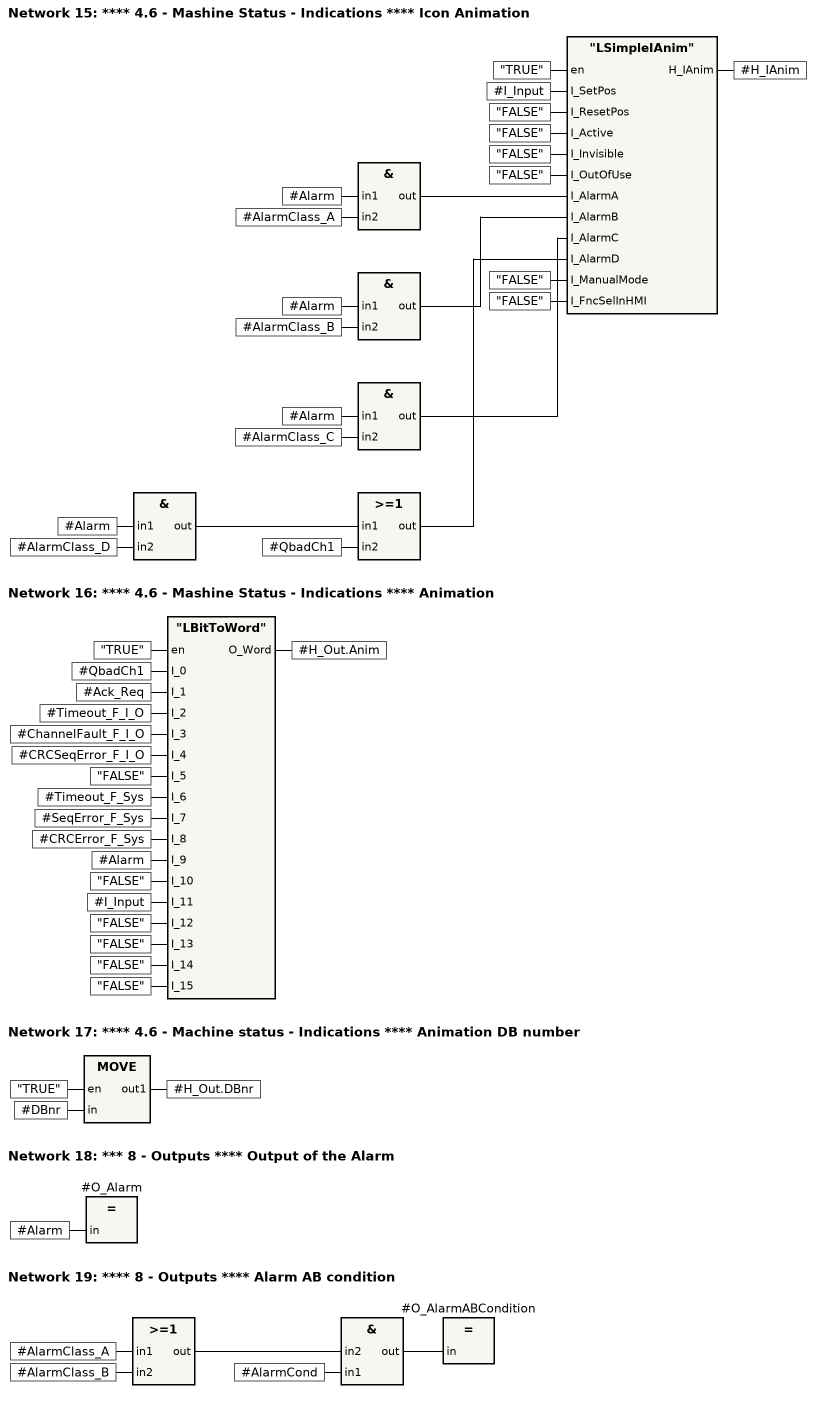
   IF "TRUE" THEN
       "LSimpleIAnim"(I_SetPos := #I_Input,
                      I_ResetPos := "FALSE",
                      I_Active := "FALSE",
                      I_Invisible := "FALSE",
                      I_OutOfUse := "FALSE",
                      I_AlarmA := #Alarm AND #AlarmClass_A,
                      I_AlarmB := #Alarm AND #AlarmClass_B,
                      I_AlarmC := #Alarm AND #AlarmClass_C,
                      I_AlarmD := (#Alarm AND #AlarmClass_D) OR #QbadCh1,
                      I_ManualMode := "FALSE",
                      I_FncSelInHMI := "FALSE",
                      H_IAnim => #H_IAnim);
   END_IF;
END_REGION

REGION Network 16: **** 4.6 - Mashine Status - Indications **** Animation
   // Animation
   IF "TRUE" THEN
       "LBitToWord"(I_0 := #QbadCh1,
                    I_1 := #Ack_Req,
                    I_2 := #Timeout_F_I_O,
                    I_3 := #ChannelFault_F_I_O,
                    I_4 := #CRCSeqError_F_I_O,
                    I_5 := "FALSE",
                    I_6 := #Timeout_F_Sys,
                    I_7 := #SeqError_F_Sys,
                    I_8 := #CRCError_F_Sys,
                    I_9 := #Alarm,
                    I_10 := "FALSE",
                    I_11 := #I_Input,
                    I_12 := "FALSE",
                    I_13 := "FALSE",
                    I_14 := "FALSE",
                    I_15 := "FALSE",
                    O_Word => #H_Out.Anim);
   END_IF;
END_REGION

REGION Network 17: **** 4.6 - Machine status - Indications **** Animation DB number
   // Animation DB number
   IF "TRUE" THEN #H_Out.DBnr := #DBnr; END_IF;
END_REGION

REGION Network 18: *** 8 - Outputs **** Output of the Alarm
   // Output of the Alarm
   #O_Alarm := #Alarm;
END_REGION

REGION Network 19: **** 8 - Outputs **** Alarm AB condition
   // Alarm AB condition
   #O_AlarmABCondition := (#AlarmClass_A OR #AlarmClass_B) AND #AlarmCond;
END_REGION
END_FUNCTION_BLOCK

FUNCTION_BLOCK "L1SafetyFbkAlarm"   // FB1422, FBD
TITLE = L1SafetyFbkAlarm
{ S7_Optimized_Access := 'FALSE' }
AUTHOR : VCC
FAMILY : AlarmHnd
NAME : 1SafeAlm
VERSION : 0.3
// ================================================================================
// TThis module evalute the diagnostic byte from the Siemens safety Functionblock 
// FB 216 "F_FDBACK" and generates a feedback alarm in the standard program.
// A boolean output is available to inform the upper level that the alarm can be 
// reset.
// This module generates also a word containing all necessary information for HMI 
// Icon animation, and a word with all information for HMI safety module 
// diagnostic screen. 
// ================================================================================
// stored: AutoNumber false, IsIECCheckEnabled false, SetENOAutomatically False, UDAEnableTagReadback false
   VAR_INPUT
      I_Feedback { ExternalAccessible := 'False'; ExternalVisible := 'False'; ExternalWritable := 'False'} : Bool;   // Input feedback
      I_AlarmClass { ExternalAccessible := 'False'; ExternalVisible := 'False'; ExternalWritable := 'False'} : Char;   // Alarm class -> A - B - C - D or E
      I_EnableAlarm { ExternalAccessible := 'False'; ExternalVisible := 'False'; ExternalWritable := 'False'} : Bool := TRUE;   // Enable alarm from upper level (0=disable/1=enable)
      I_AlarmResetPB { ExternalAccessible := 'False'; ExternalVisible := 'False'; ExternalWritable := 'False'} : Bool;   // Alarm reset pushbutton is activated
      I_SafetyCard_DIAG { ExternalAccessible := 'False'; ExternalVisible := 'False'; ExternalWritable := 'False'} : Byte;   // Automatically generated DB from F-Modul (F-Peripherie DB)
   END_VAR
   VAR_OUTPUT
      O_Alarm { ExternalAccessible := 'False'; ExternalVisible := 'False'; ExternalWritable := 'False'} : Bool;   // Alarm
      O_AlarmABCondiion { ExternalAccessible := 'False'; ExternalVisible := 'False'; ExternalWritable := 'False'} : Bool;   // Alarm AB condition
      H_IAnim { ExternalAccessible := 'False'; ExternalVisible := 'False'; ExternalWritable := 'False'} : Word;   // Icon Animation
   END_VAR
   VAR DB_SPECIFIC
      H_Out : Struct   // HMI
         Anim : Word;   // HMI Animation of the object
         DBnr : Int;   // HMI Animation DB number
      END_STRUCT;
      FeedbackError { ExternalAccessible := 'False'; ExternalVisible := 'False'; ExternalWritable := 'False'} : Bool;   // Feedback error or incorrect feedback time setting (= state of ERROR)
      Passivation { ExternalAccessible := 'False'; ExternalVisible := 'False'; ExternalWritable := 'False'} : Bool;   // Passivation of F-I/O/channel controlled by output Q
      ErrorSignal0 { ExternalAccessible := 'False'; ExternalVisible := 'False'; ExternalWritable := 'False'} : Bool;   // After feedback error: feedback input has permanent signal state of 0
      ErrorSignal1 { ExternalAccessible := 'False'; ExternalVisible := 'False'; ExternalWritable := 'False'} : Bool;   // For feedback error: input ACK has a permanent signal state of 1
      AckReq { ExternalAccessible := 'False'; ExternalVisible := 'False'; ExternalWritable := 'False'} : Bool;   // Acknowledgement required (= state of ACK_REQ)
      Q { ExternalAccessible := 'False'; ExternalVisible := 'False'; ExternalWritable := 'False'} : Bool;   // State of output Q
      Alarm { ExternalAccessible := 'False'; ExternalVisible := 'False'; ExternalWritable := 'False'} : Bool;   // Alarm
      AlarmClass_A { ExternalAccessible := 'False'; ExternalVisible := 'False'; ExternalWritable := 'False'} : Bool;   // The alarm is from alarm class A
      AlarmClass_B { ExternalAccessible := 'False'; ExternalVisible := 'False'; ExternalWritable := 'False'} : Bool;   // The alarm is from alarm class B
      AlarmClass_C { ExternalAccessible := 'False'; ExternalVisible := 'False'; ExternalWritable := 'False'} : Bool;   // The alarm is from alarm class C
      AlarmClass_D { ExternalAccessible := 'False'; ExternalVisible := 'False'; ExternalWritable := 'False'} : Bool;   // The alarm is from alarm class D
      AlarmCond { ExternalAccessible := 'False'; ExternalVisible := 'False'; ExternalWritable := 'False'} : Bool;   // Alarm condition
      DBnr { ExternalAccessible := 'False'; ExternalVisible := 'False'; ExternalWritable := 'False'} : Int;   // HMI DB number
   END_VAR
BEGIN

NETWORK
TITLE = **** 1 - Inputs **** DB number
// DB number
      L     DINO;
      T     #DBnr;

NETWORK
TITLE = **** 1 - Inputs **** Alarm class
// Alarm class
// Alarm class = D
      L     #I_AlarmClass;
      L     'D';
      ==I;
      =     #AlarmClass_D;

// Alarm class = C
      L     #I_AlarmClass;
      L     'C';
      ==I;
      =     #AlarmClass_C;

// Alarm class = B
      L     #I_AlarmClass;
      L     'B';
      ==I;
      =     #AlarmClass_B;

// Alarm class = A
      AN    #AlarmClass_B;
      AN    #AlarmClass_C;
      AN    #AlarmClass_D;
      =     #AlarmClass_A;


REGION Network 3: **** 1 - Inputs **** Feedback error or incorrect feedback time setting (= state of ERROR)
   // Feedback error or incorrect feedback time setting (= state of ERROR)
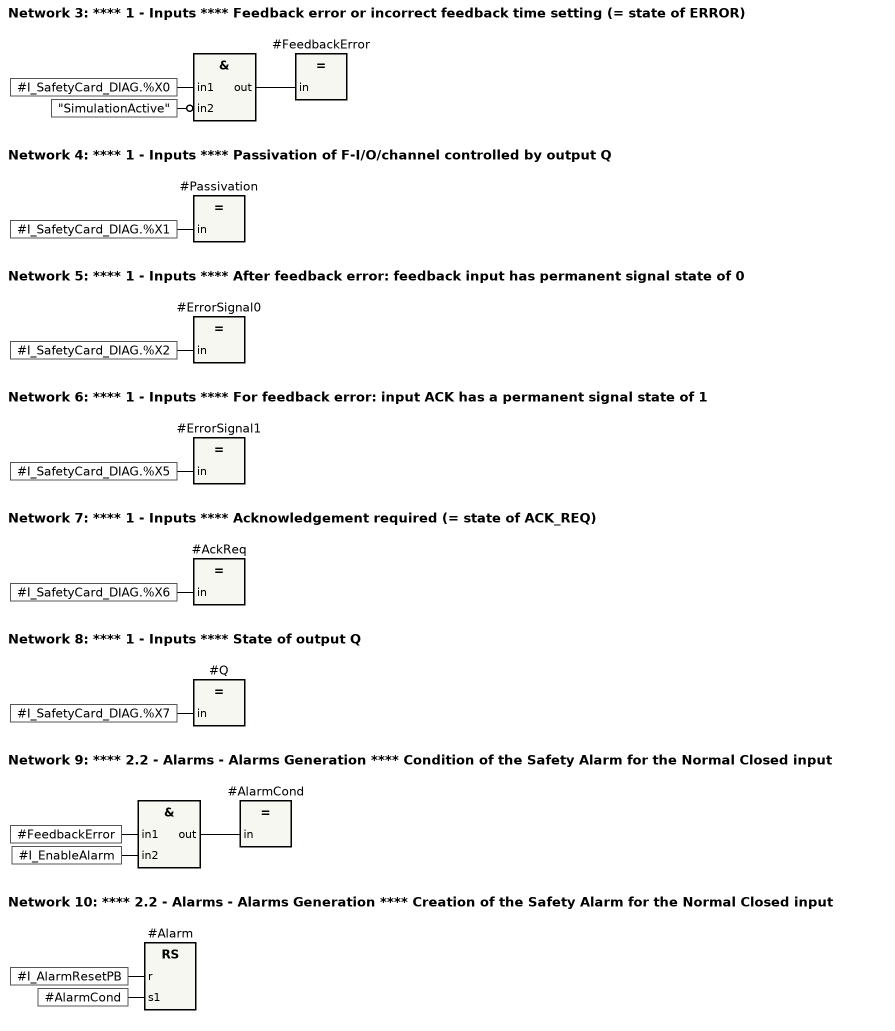
   #FeedbackError := #I_SafetyCard_DIAG.%X0 AND NOT "SimulationActive";
END_REGION

REGION Network 4: **** 1 - Inputs **** Passivation of F-I/O/channel controlled by output Q
   // Passivation of F-I/O/channel controlled by output Q
   #Passivation := #I_SafetyCard_DIAG.%X1;
END_REGION

REGION Network 5: **** 1 - Inputs **** After feedback error: feedback input has permanent signal state of 0
   // After feedback error: feedback input has permanent signal state of 0
   #ErrorSignal0 := #I_SafetyCard_DIAG.%X2;
END_REGION

REGION Network 6: **** 1 - Inputs **** For feedback error: input ACK has a permanent signal state of 1
   // For feedback error: input ACK has a permanent signal state of 1
   #ErrorSignal1 := #I_SafetyCard_DIAG.%X5;
END_REGION

REGION Network 7: **** 1 - Inputs **** Acknowledgement required (= state of ACK_REQ)
   // Acknowledgement required (= state of ACK_REQ)
   #AckReq := #I_SafetyCard_DIAG.%X6;
END_REGION

REGION Network 8: **** 1 - Inputs **** State of output Q
   // State of output Q
   #Q := #I_SafetyCard_DIAG.%X7;
END_REGION

REGION Network 9: **** 2.2 - Alarms - Alarms Generation **** Condition of the Safety Alarm for the Normal Closed input
   // Condition of the Safety Alarm for the Normal Closed input
   #AlarmCond := #FeedbackError AND #I_EnableAlarm;
END_REGION

REGION Network 10: **** 2.2 - Alarms - Alarms Generation **** Creation of the Safety Alarm for the Normal Closed input
   // Creation of the Safety Alarm for the Normal Closed input
   IF #I_AlarmResetPB THEN
       #Alarm := FALSE;   // RS flip-flop
   END_IF;
   IF #AlarmCond THEN #Alarm := TRUE; END_IF;
END_REGION

REGION Network 11: **** 4.6 - Mashine Status - Indications **** Icon Animation
   // Icon Animation
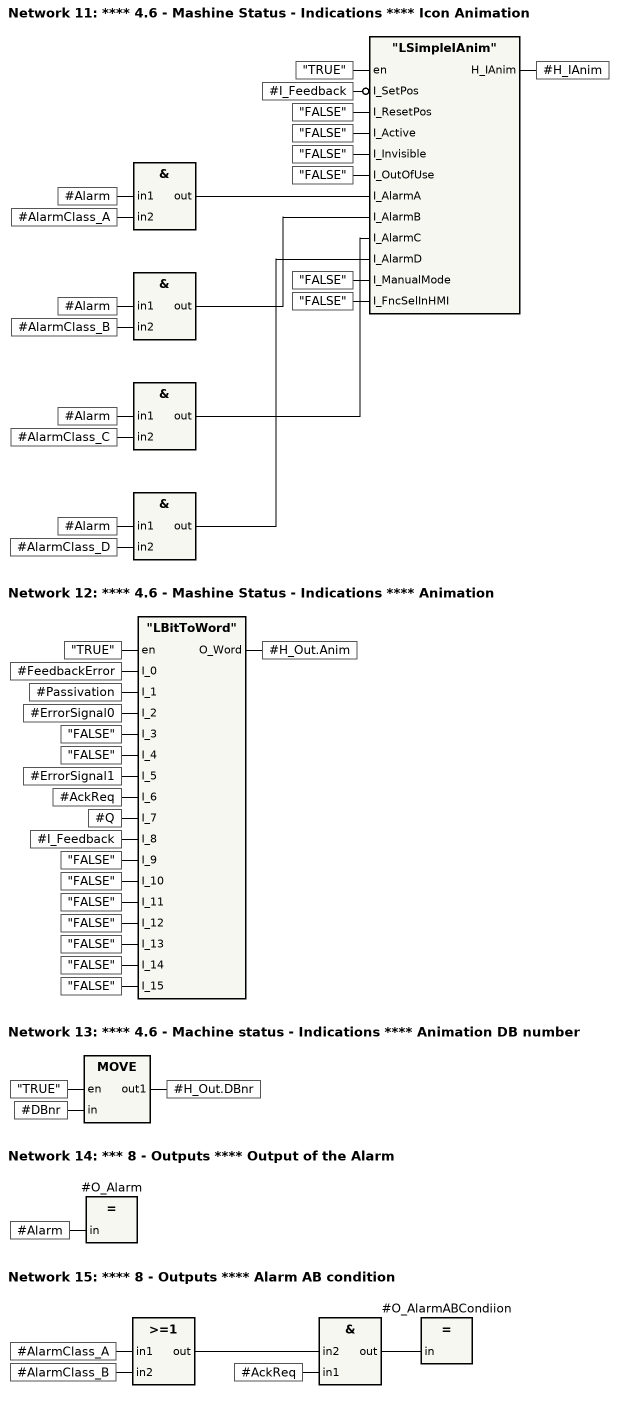
   IF "TRUE" THEN
       "LSimpleIAnim"(I_SetPos := NOT #I_Feedback,
                      I_ResetPos := "FALSE",
                      I_Active := "FALSE",
                      I_Invisible := "FALSE",
                      I_OutOfUse := "FALSE",
                      I_AlarmA := #Alarm AND #AlarmClass_A,
                      I_AlarmB := #Alarm AND #AlarmClass_B,
                      I_AlarmC := #Alarm AND #AlarmClass_C,
                      I_AlarmD := #Alarm AND #AlarmClass_D,
                      I_ManualMode := "FALSE",
                      I_FncSelInHMI := "FALSE",
                      H_IAnim => #H_IAnim);
   END_IF;
END_REGION

REGION Network 12: **** 4.6 - Mashine Status - Indications **** Animation
   // Animation
   IF "TRUE" THEN
       "LBitToWord"(I_0 := #FeedbackError,
                    I_1 := #Passivation,
                    I_2 := #ErrorSignal0,
                    I_3 := "FALSE",
                    I_4 := "FALSE",
                    I_5 := #ErrorSignal1,
                    I_6 := #AckReq,
                    I_7 := #Q,
                    I_8 := #I_Feedback,
                    I_9 := "FALSE",
                    I_10 := "FALSE",
                    I_11 := "FALSE",
                    I_12 := "FALSE",
                    I_13 := "FALSE",
                    I_14 := "FALSE",
                    I_15 := "FALSE",
                    O_Word => #H_Out.Anim);
   END_IF;
END_REGION

REGION Network 13: **** 4.6 - Machine status - Indications **** Animation DB number
   // Animation DB number
   IF "TRUE" THEN #H_Out.DBnr := #DBnr; END_IF;
END_REGION

REGION Network 14: *** 8 - Outputs **** Output of the Alarm
   // Output of the Alarm
   #O_Alarm := #Alarm;
END_REGION

REGION Network 15: **** 8 - Outputs **** Alarm AB condition
   // Alarm AB condition
   #O_AlarmABCondiion := (#AlarmClass_A OR #AlarmClass_B) AND #AckReq;
END_REGION
END_FUNCTION_BLOCK

FUNCTION_BLOCK "L1AlarmDly"   // FB1423, FBD
TITLE = L1AlarmDly
{ S7_Optimized_Access := 'FALSE' }
AUTHOR : VCC
FAMILY : AlarmHnd
NAME : 1AlarmDl
VERSION : 0.1
// ================================================================================
// This module is used everywhere one alarm shall be generated when one (security) 
// input becomes True. The alarm have a delay time set in millieseconds.
// The alarm can be True only when the input Enable Alarm is also True.
// The alarm can be True only when the input Disable Alarm is False. When the 
// alarm is disable from HMI, a boolean output is available to inform the upper 
// level and do action in the Alarm summary.
// When the conditions to generate the alarm is disappear, a boolean output is 
// available to inform the upper level that the alarm can be reset.
// The alarm is reset by means of the AlarmResetPB signal.
// ================================================================================
// stored: AutoNumber false, IsIECCheckEnabled false, SetENOAutomatically False, UDAEnableTagReadback false
   VAR_INPUT
      I_Input { ExternalAccessible := 'False'; ExternalVisible := 'False'; ExternalWritable := 'False'} : Bool;   // Input signal of the alarm
      I_AlarmClass { ExternalAccessible := 'False'; ExternalVisible := 'False'; ExternalWritable := 'False'} : Char;   // Alarm class -> A - B - C - D or E
      I_EnableAlarm { ExternalAccessible := 'False'; ExternalVisible := 'False'; ExternalWritable := 'False'} : Bool := TRUE;   // Enable alarm from upper level
      I_AlarmResetPB { ExternalAccessible := 'False'; ExternalVisible := 'False'; ExternalWritable := 'False'} : Bool;   // Alarm reset pushbutton is activated
      I_Invisible { ExternalAccessible := 'False'; ExternalVisible := 'False'; ExternalWritable := 'False'} : Bool;   // Invisible
      C_NcAlarm { ExternalAccessible := 'False'; ExternalVisible := 'False'; ExternalWritable := 'False'} : Bool;   // Normally closed contact
   END_VAR
   VAR_OUTPUT
      O_Alarm { ExternalAccessible := 'False'; ExternalVisible := 'False'; ExternalWritable := 'False'} : Bool;   // Alarm
      O_AlarmDly { ExternalAccessible := 'False'; ExternalVisible := 'False'; ExternalWritable := 'False'} : Bool;   // Alarm delayed
      O_AlarmABCondition { ExternalAccessible := 'False'; ExternalVisible := 'False'; ExternalWritable := 'False'} : Bool;   // Alarm AB condition
      H_IAnim { ExternalAccessible := 'False'; ExternalVisible := 'False'; ExternalWritable := 'False'} : Word;   // Icon animation
   END_VAR
   VAR DB_SPECIFIC
      H_In : Struct   // HMI
         DelayTime : DInt;   // Delay time in millieseconds
      END_STRUCT;
      H_Out : Struct   // HMI
         Anim : Word;   // HMI Animation of the object
         DBnr : Int;   // HMI Animation DB number
      END_STRUCT;
      Alarm : Bool;   // Alarm
      AlarmDly : Bool;   // Alarm delayed
      AlarmClass_A { ExternalAccessible := 'False'; ExternalVisible := 'False'; ExternalWritable := 'False'} : Bool;   // The alarm is from alarm class A
      AlarmClass_B { ExternalAccessible := 'False'; ExternalVisible := 'False'; ExternalWritable := 'False'} : Bool;   // The alarm is from alarm class B
      AlarmClass_C { ExternalAccessible := 'False'; ExternalVisible := 'False'; ExternalWritable := 'False'} : Bool;   // The alarm is from alarm class C
      AlarmClass_D { ExternalAccessible := 'False'; ExternalVisible := 'False'; ExternalWritable := 'False'} : Bool;   // The alarm is from alarm class D
      AlarmClass_E { ExternalAccessible := 'False'; ExternalVisible := 'False'; ExternalWritable := 'False'} : Bool;   // The alarm is from alarm class E
      AlarmCond : Bool;   // Alarm condition
      InputCond : Bool;   // Input condition to set the alarm
      DBnr { ExternalAccessible := 'False'; ExternalVisible := 'False'; ExternalWritable := 'False'} : Int;   // HMI DB number
   END_VAR
   VAR
      AlarmDlyTimer { S7_SetPoint := 'True'} : "LTimer";   // Timer for delayed alarm
   END_VAR
BEGIN

NETWORK
TITLE = **** 1 - Inputs **** DB number
// DB number
      L     DINO;
      T     #DBnr;

NETWORK
TITLE = **** 1 - Inputs **** Alarm class
// Alarm class
// Alarm class = E
      L     #I_AlarmClass;
      L     'E';
      ==I;
      =     #AlarmClass_E;

// Alarm class = D
      L     #I_AlarmClass;
      L     'D';
      ==I;
      =     #AlarmClass_D;

// Alarm class = C
      L     #I_AlarmClass;
      L     'C';
      ==I;
      =     #AlarmClass_C;

// Alarm class = B
      L     #I_AlarmClass;
      L     'B';
      ==I;
      =     #AlarmClass_B;

// Alarm class = A
      AN    #AlarmClass_B;
      AN    #AlarmClass_C;
      AN    #AlarmClass_D;
      AN    #AlarmClass_E;
      =     #AlarmClass_A;


REGION Network 3: **** 1 - Inputs **** Input condition
   // Input condition
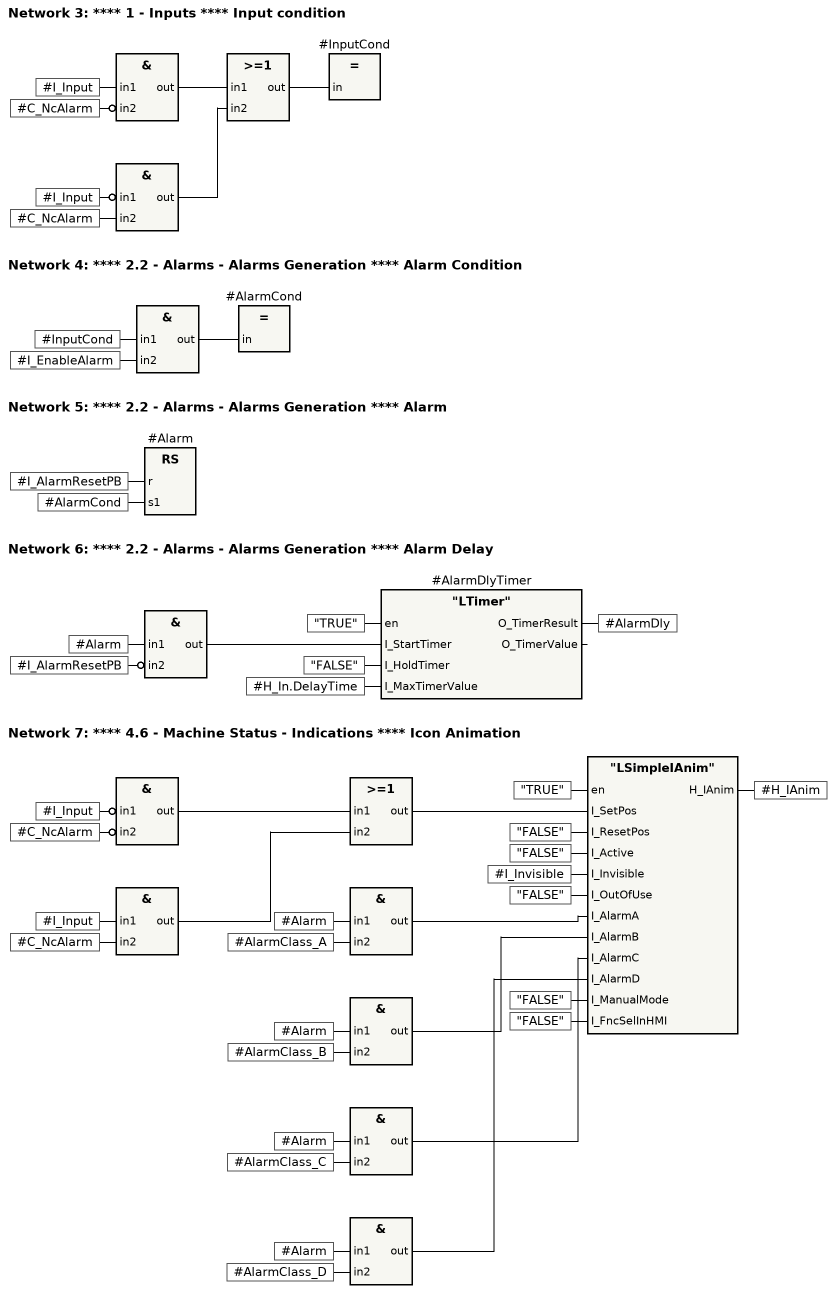
   #InputCond := (#I_Input AND NOT #C_NcAlarm) OR (NOT #I_Input AND #C_NcAlarm);
END_REGION

REGION Network 4: **** 2.2 - Alarms - Alarms Generation **** Alarm Condition
   // Condition of the Alarm
   #AlarmCond := #InputCond AND #I_EnableAlarm;
END_REGION

REGION Network 5: **** 2.2 - Alarms - Alarms Generation **** Alarm
   // Creation of the Alarm
   IF #I_AlarmResetPB THEN
       #Alarm := FALSE;   // RS flip-flop
   END_IF;
   IF #AlarmCond THEN #Alarm := TRUE; END_IF;
END_REGION

REGION Network 6: **** 2.2 - Alarms - Alarms Generation **** Alarm Delay
   // Creation of the delayed Alarm
   IF "TRUE" THEN
       #AlarmDlyTimer(I_StartTimer := #Alarm AND NOT #I_AlarmResetPB,   // "LTimer"
                      I_HoldTimer := "FALSE",
                      I_MaxTimerValue := #H_In.DelayTime,
                      O_TimerResult => #AlarmDly);
   END_IF;
END_REGION

REGION Network 7: **** 4.6 - Machine Status - Indications **** Icon Animation
   // Icon Animation
   IF "TRUE" THEN
       "LSimpleIAnim"(I_SetPos := (NOT #I_Input AND NOT #C_NcAlarm) OR (#I_Input AND #C_NcAlarm),
                      I_ResetPos := "FALSE",
                      I_Active := "FALSE",
                      I_Invisible := #I_Invisible,
                      I_OutOfUse := "FALSE",
                      I_AlarmA := #Alarm AND #AlarmClass_A,
                      I_AlarmB := #Alarm AND #AlarmClass_B,
                      I_AlarmC := #Alarm AND #AlarmClass_C,
                      I_AlarmD := #Alarm AND #AlarmClass_D,
                      I_ManualMode := "FALSE",
                      I_FncSelInHMI := "FALSE",
                      H_IAnim => #H_IAnim);
   END_IF;
END_REGION

REGION Network 8: **** 4.6 - Machine Status - Indications **** Animation
   // Animation
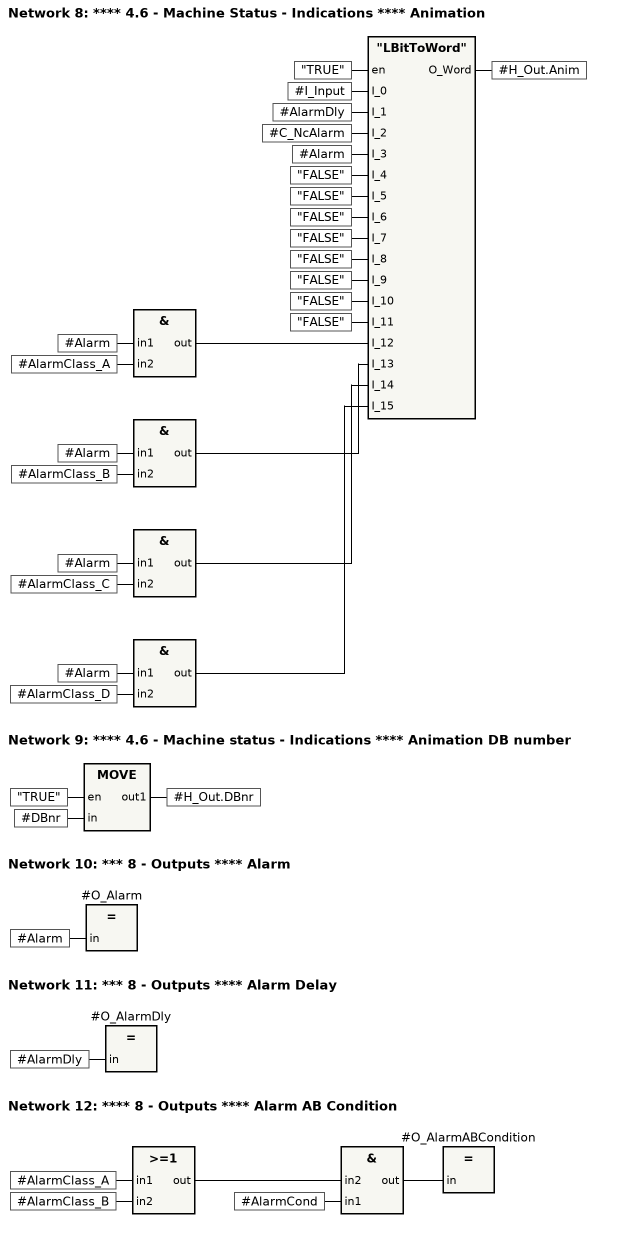
   IF "TRUE" THEN
       "LBitToWord"(I_0 := #I_Input,
                    I_1 := #AlarmDly,
                    I_2 := #C_NcAlarm,
                    I_3 := #Alarm,
                    I_4 := "FALSE",
                    I_5 := "FALSE",
                    I_6 := "FALSE",
                    I_7 := "FALSE",
                    I_8 := "FALSE",
                    I_9 := "FALSE",
                    I_10 := "FALSE",
                    I_11 := "FALSE",
                    I_12 := #Alarm AND #AlarmClass_A,
                    I_13 := #Alarm AND #AlarmClass_B,
                    I_14 := #Alarm AND #AlarmClass_C,
                    I_15 := #Alarm AND #AlarmClass_D,
                    O_Word => #H_Out.Anim);
   END_IF;
END_REGION

REGION Network 9: **** 4.6 - Machine status - Indications **** Animation DB number
   IF "TRUE" THEN #H_Out.DBnr := #DBnr; END_IF;
END_REGION

REGION Network 10: *** 8 - Outputs **** Alarm
   // Output of the Alarm
   #O_Alarm := #Alarm;
END_REGION

REGION Network 11: *** 8 - Outputs **** Alarm Delay
   // Output of the Alarm
   #O_AlarmDly := #AlarmDly;
END_REGION

REGION Network 12: **** 8 - Outputs **** Alarm AB Condition
   // Alarm AB condition
   #O_AlarmABCondition := (#AlarmClass_A OR #AlarmClass_B) AND #AlarmCond;
END_REGION
END_FUNCTION_BLOCK

FUNCTION_BLOCK "L2Alarm"   // FB1425, FBD
TITLE = L2Alarm
{ S7_Optimized_Access := 'FALSE' }
AUTHOR : VCC
FAMILY : AlarmHnd
NAME : 2Alarm
VERSION : 1.0
// ================================================================================
// This module is used everywhere two alarms shall be generated from one object.
// The alarm can be True only when the input Enable Alarm is also True.
// The alarm can be True only when the input Disable Alarm is False. When the 
// alarm is disable from HMI, a boolean output is available to inform the upper 
// level and do action in the Alarm summary.
// When the conditions to generate the alarm is disappear, a boolean output is 
// available to inform the upper level that the alarm can be reset.
// ================================================================================
// stored: AutoNumber false, IsIECCheckEnabled false, SetENOAutomatically False, UDAEnableTagReadback false
   VAR_INPUT
      I_Input1 { ExternalAccessible := 'False'; ExternalVisible := 'False'; ExternalWritable := 'False'} : Bool;   // Input signal 1 of the alarm
      I_AlarmClass1 { ExternalAccessible := 'False'; ExternalVisible := 'False'; ExternalWritable := 'False'} : Char;   // Alarm class -> A - B - C - D or E
      I_Input2 { ExternalAccessible := 'False'; ExternalVisible := 'False'; ExternalWritable := 'False'} : Bool;   // Input signal 2 of the alarm
      I_AlarmClass2 { ExternalAccessible := 'False'; ExternalVisible := 'False'; ExternalWritable := 'False'} : Char;   // Alarm class -> A - B - C - D or E
      I_EnableAlarm { ExternalAccessible := 'False'; ExternalVisible := 'False'; ExternalWritable := 'False'} : Bool := TRUE;   // Enable alarm from upper level
      I_AlarmResetPB { ExternalAccessible := 'False'; ExternalVisible := 'False'; ExternalWritable := 'False'} : Bool;   // Alarm reset pushbutton is activated
      I_Invisible { ExternalAccessible := 'False'; ExternalVisible := 'False'; ExternalWritable := 'False'} : Bool;   // Invisible
      C_NcAlarm { ExternalAccessible := 'False'; ExternalVisible := 'False'; ExternalWritable := 'False'} : Bool;   // Alarm contact NC
   END_VAR
   VAR_OUTPUT
      O_Alarm1 { ExternalAccessible := 'False'; ExternalVisible := 'False'; ExternalWritable := 'False'} : Bool;   // Alarm 1
      O_Alarm2 { ExternalAccessible := 'False'; ExternalVisible := 'False'; ExternalWritable := 'False'} : Bool;   // Alarm 2
      O_AlarmDisabled { ExternalAccessible := 'False'; ExternalVisible := 'False'; ExternalWritable := 'False'} : Bool;   // Alarm disabled from HMI
      O_AlarmABCondition { ExternalAccessible := 'False'; ExternalVisible := 'False'; ExternalWritable := 'False'} : Bool;   // Alarm AB condition
      H_IAnim1 { ExternalAccessible := 'False'; ExternalVisible := 'False'; ExternalWritable := 'False'} : Word;   // Icon Animation
      H_IAnim2 { ExternalAccessible := 'False'; ExternalVisible := 'False'; ExternalWritable := 'False'} : Word;   // Icon Animation
   END_VAR
   VAR DB_SPECIFIC
      H_In : Struct   // HMI
         DisableAlarm : Bool;   // Disable alarm from HMI
      END_STRUCT;
      H_Out : Struct   // HMI
         Anim1 : Word;   // HMI Animation of the object
         Anim2 : Word;   // HMI Animation of the object
         DBnr : Int;   // HMI Animation DB number
      END_STRUCT;
      Alarm1 { ExternalAccessible := 'False'; ExternalVisible := 'False'; ExternalWritable := 'False'} : Bool;   // Alarm 1
      AlarmClass1_A { ExternalAccessible := 'False'; ExternalVisible := 'False'; ExternalWritable := 'False'} : Bool;   // The alarm is from alarm class A
      AlarmClass1_B { ExternalAccessible := 'False'; ExternalVisible := 'False'; ExternalWritable := 'False'} : Bool;   // The alarm is from alarm class B
      AlarmClass1_C { ExternalAccessible := 'False'; ExternalVisible := 'False'; ExternalWritable := 'False'} : Bool;   // The alarm is from alarm class C
      AlarmClass1_D { ExternalAccessible := 'False'; ExternalVisible := 'False'; ExternalWritable := 'False'} : Bool;   // The alarm is from alarm class D
      AlarmClass1_E { ExternalAccessible := 'False'; ExternalVisible := 'False'; ExternalWritable := 'False'} : Bool;   // The alarm is from alarm class E
      AlarmCond1 { ExternalAccessible := 'False'; ExternalVisible := 'False'; ExternalWritable := 'False'} : Bool;   // Alarm condition 1
      Alarm2 { ExternalAccessible := 'False'; ExternalVisible := 'False'; ExternalWritable := 'False'} : Bool;   // Alarm 2
      AlarmClass2_A { ExternalAccessible := 'False'; ExternalVisible := 'False'; ExternalWritable := 'False'} : Bool;   // The alarm is from alarm class A
      AlarmClass2_B { ExternalAccessible := 'False'; ExternalVisible := 'False'; ExternalWritable := 'False'} : Bool;   // The alarm is from alarm class B
      AlarmClass2_C { ExternalAccessible := 'False'; ExternalVisible := 'False'; ExternalWritable := 'False'} : Bool;   // The alarm is from alarm class C
      AlarmClass2_D { ExternalAccessible := 'False'; ExternalVisible := 'False'; ExternalWritable := 'False'} : Bool;   // The alarm is from alarm class D
      AlarmClass2_E { ExternalAccessible := 'False'; ExternalVisible := 'False'; ExternalWritable := 'False'} : Bool;   // The alarm is from alarm class E
      AlarmCond2 { ExternalAccessible := 'False'; ExternalVisible := 'False'; ExternalWritable := 'False'} : Bool;   // Alarm condition 2
      DBnr { ExternalAccessible := 'False'; ExternalVisible := 'False'; ExternalWritable := 'False'} : Int;   // HMI DB number
   END_VAR
BEGIN

NETWORK
TITLE = **** 1 - Inputs **** DB number
// DB number
      L     DINO;
      T     #DBnr;

NETWORK
TITLE = **** 1 - Inputs **** Alarm class 1
// Alarm class
// Alarm class = E
      L     #I_AlarmClass1;
      L     'E';
      ==I;
      =     #AlarmClass1_E;

// Alarm class = D
      L     #I_AlarmClass1;
      L     'D';
      ==I;
      =     #AlarmClass1_D;

// Alarm class = C
      L     #I_AlarmClass1;
      L     'C';
      ==I;
      =     #AlarmClass1_C;

// Alarm class = B
      L     #I_AlarmClass1;
      L     'B';
      ==I;
      =     #AlarmClass1_B;

// Alarm class = A
      AN    #AlarmClass1_B;
      AN    #AlarmClass1_C;
      AN    #AlarmClass1_D;
      AN    #AlarmClass1_E;
      =     #AlarmClass1_A;


NETWORK
TITLE = **** 1 - Inputs **** Alarm class 2
// Alarm class
// Alarm class = E
      L     #I_AlarmClass2;
      L     'E';
      ==I;
      =     #AlarmClass2_E;

// Alarm class = D
      L     #I_AlarmClass2;
      L     'D';
      ==I;
      =     #AlarmClass2_D;

// Alarm class = C
      L     #I_AlarmClass2;
      L     'C';
      ==I;
      =     #AlarmClass2_C;

// Alarm class = B
      L     #I_AlarmClass2;
      L     'B';
      ==I;
      =     #AlarmClass2_B;

// Alarm class = A
      AN    #AlarmClass2_B;
      AN    #AlarmClass2_C;
      AN    #AlarmClass2_D;
      AN    #AlarmClass2_E;
      =     #AlarmClass2_A;


REGION Network 4: **** 2.2 - Alarms - Alarms Generation **** Alarm Condition 1
   // Condition of Alarm 1
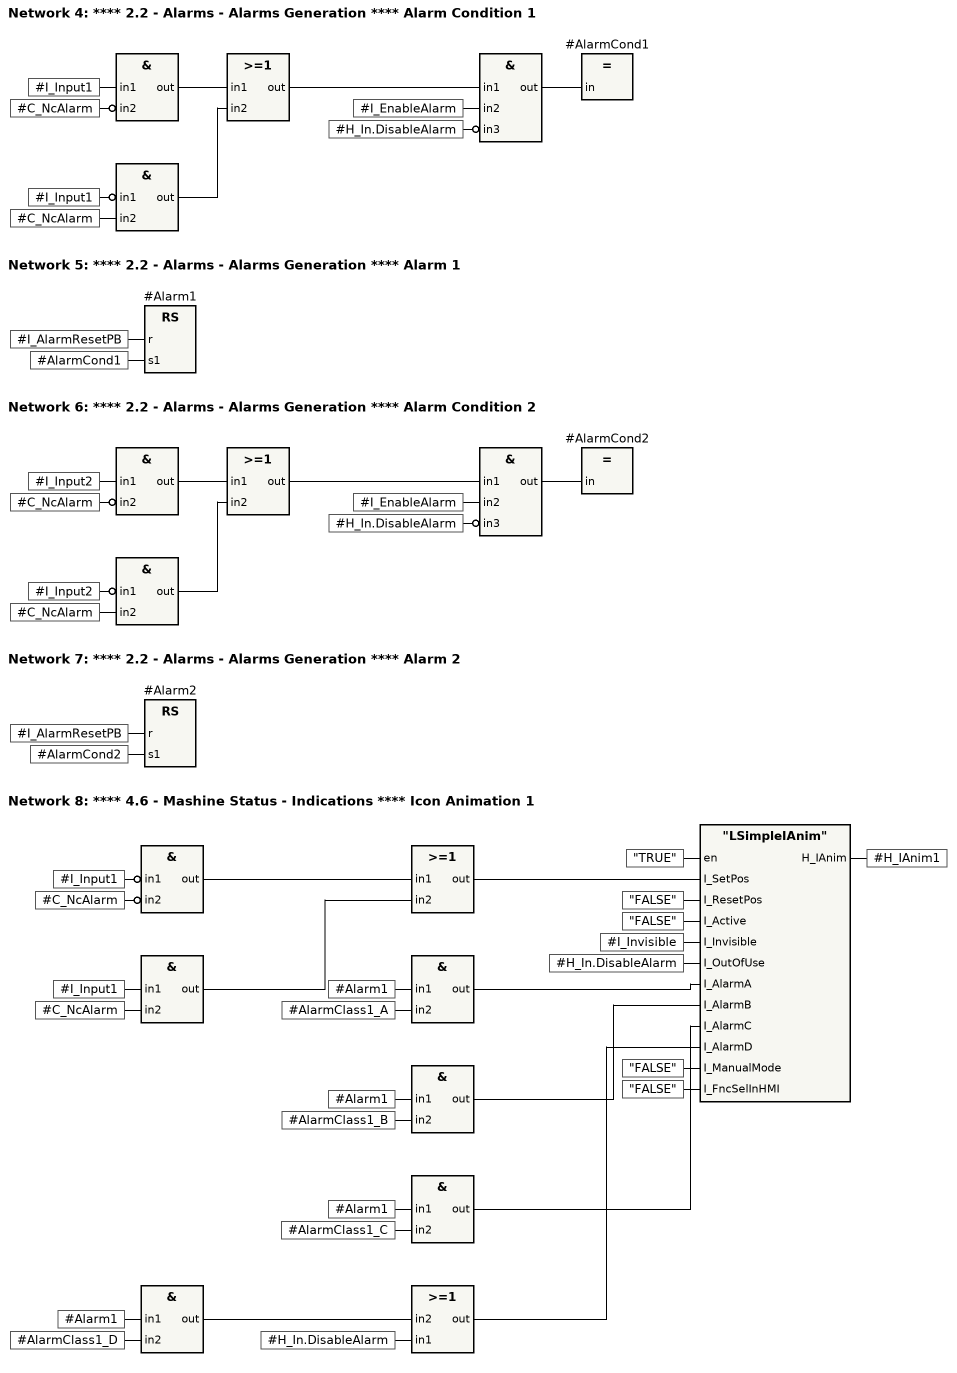
   #AlarmCond1 := ((#I_Input1 AND NOT #C_NcAlarm) OR (NOT #I_Input1 AND #C_NcAlarm)) AND #I_EnableAlarm AND NOT #H_In.DisableAlarm;
END_REGION

REGION Network 5: **** 2.2 - Alarms - Alarms Generation **** Alarm 1
   // Creation of Alarm 1
   IF #I_AlarmResetPB THEN
       #Alarm1 := FALSE;   // RS flip-flop
   END_IF;
   IF #AlarmCond1 THEN #Alarm1 := TRUE; END_IF;
END_REGION

REGION Network 6: **** 2.2 - Alarms - Alarms Generation **** Alarm Condition 2
   // Condition of Alarm 2
   #AlarmCond2 := ((#I_Input2 AND NOT #C_NcAlarm) OR (NOT #I_Input2 AND #C_NcAlarm)) AND #I_EnableAlarm AND NOT #H_In.DisableAlarm;
END_REGION

REGION Network 7: **** 2.2 - Alarms - Alarms Generation **** Alarm 2
   // Creation of Alarm 2
   IF #I_AlarmResetPB THEN
       #Alarm2 := FALSE;   // RS flip-flop
   END_IF;
   IF #AlarmCond2 THEN #Alarm2 := TRUE; END_IF;
END_REGION

REGION Network 8: **** 4.6 - Mashine Status - Indications **** Icon Animation 1
   // Icon Animation 1
   IF "TRUE" THEN
       "LSimpleIAnim"(I_SetPos := (NOT #I_Input1 AND NOT #C_NcAlarm) OR (#I_Input1 AND #C_NcAlarm),
                      I_ResetPos := "FALSE",
                      I_Active := "FALSE",
                      I_Invisible := #I_Invisible,
                      I_OutOfUse := #H_In.DisableAlarm,
                      I_AlarmA := #Alarm1 AND #AlarmClass1_A,
                      I_AlarmB := #Alarm1 AND #AlarmClass1_B,
                      I_AlarmC := #Alarm1 AND #AlarmClass1_C,
                      I_AlarmD := (#Alarm1 AND #AlarmClass1_D) OR #H_In.DisableAlarm,
                      I_ManualMode := "FALSE",
                      I_FncSelInHMI := "FALSE",
                      H_IAnim => #H_IAnim1);
   END_IF;
END_REGION

REGION Network 9: **** 4.6 - Mashine Status - Indications **** Icon Animation 2
   // Icon Animation 2
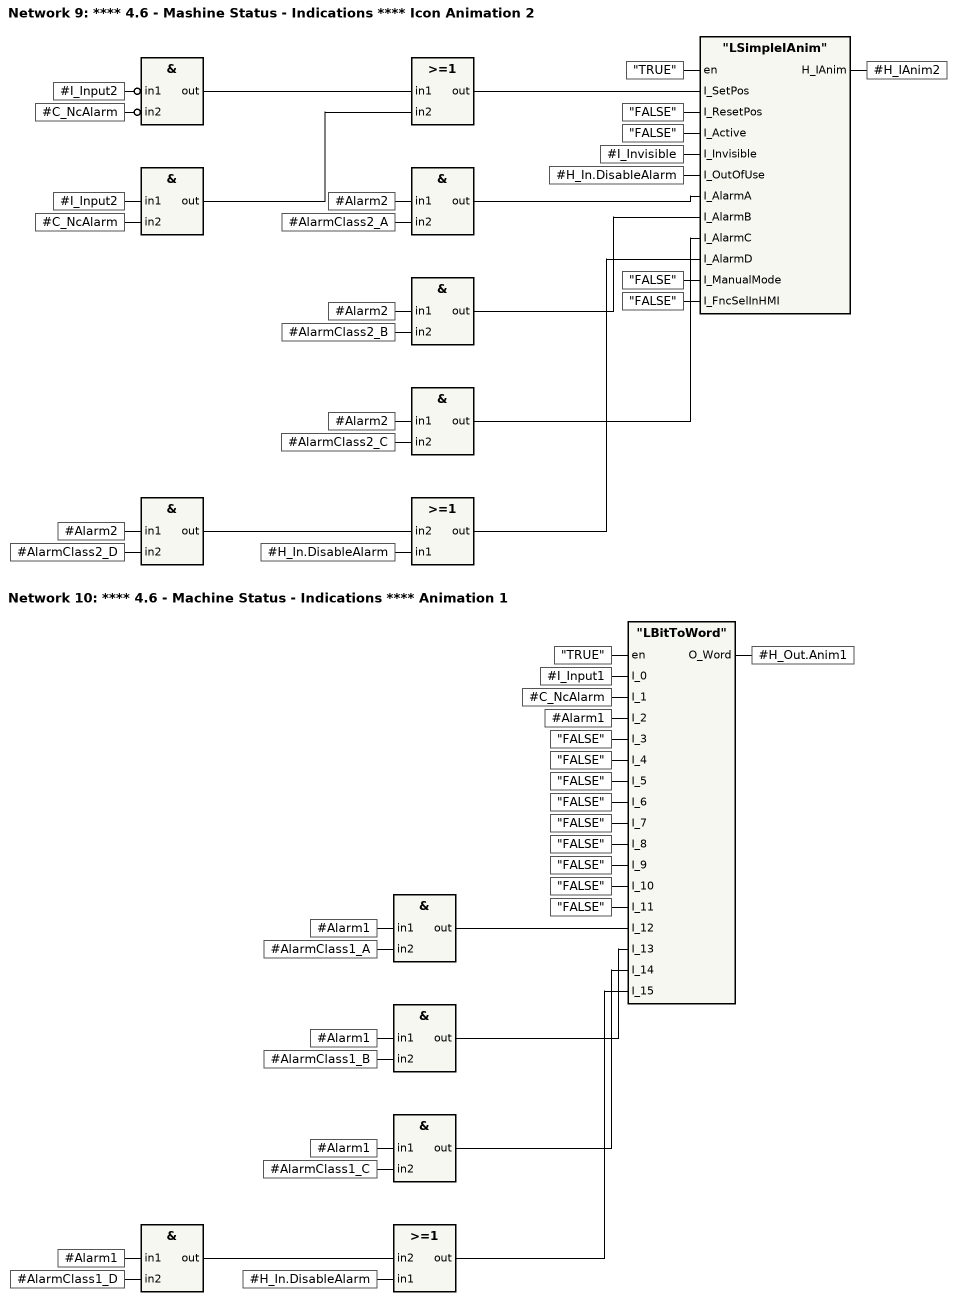
   IF "TRUE" THEN
       "LSimpleIAnim"(I_SetPos := (NOT #I_Input2 AND NOT #C_NcAlarm) OR (#I_Input2 AND #C_NcAlarm),
                      I_ResetPos := "FALSE",
                      I_Active := "FALSE",
                      I_Invisible := #I_Invisible,
                      I_OutOfUse := #H_In.DisableAlarm,
                      I_AlarmA := #Alarm2 AND #AlarmClass2_A,
                      I_AlarmB := #Alarm2 AND #AlarmClass2_B,
                      I_AlarmC := #Alarm2 AND #AlarmClass2_C,
                      I_AlarmD := (#Alarm2 AND #AlarmClass2_D) OR #H_In.DisableAlarm,
                      I_ManualMode := "FALSE",
                      I_FncSelInHMI := "FALSE",
                      H_IAnim => #H_IAnim2);
   END_IF;
END_REGION

REGION Network 10: **** 4.6 - Machine Status - Indications **** Animation 1
   // Animation 1
   IF "TRUE" THEN
       "LBitToWord"(I_0 := #I_Input1,
                    I_1 := #C_NcAlarm,
                    I_2 := #Alarm1,
                    I_3 := "FALSE",
                    I_4 := "FALSE",
                    I_5 := "FALSE",
                    I_6 := "FALSE",
                    I_7 := "FALSE",
                    I_8 := "FALSE",
                    I_9 := "FALSE",
                    I_10 := "FALSE",
                    I_11 := "FALSE",
                    I_12 := #Alarm1 AND #AlarmClass1_A,
                    I_13 := #Alarm1 AND #AlarmClass1_B,
                    I_14 := #Alarm1 AND #AlarmClass1_C,
                    I_15 := (#Alarm1 AND #AlarmClass1_D) OR #H_In.DisableAlarm,
                    O_Word => #H_Out.Anim1);
   END_IF;
END_REGION

REGION Network 11: **** 4.6 - Machine Status - Indications **** Animation 2
   // Animation 2
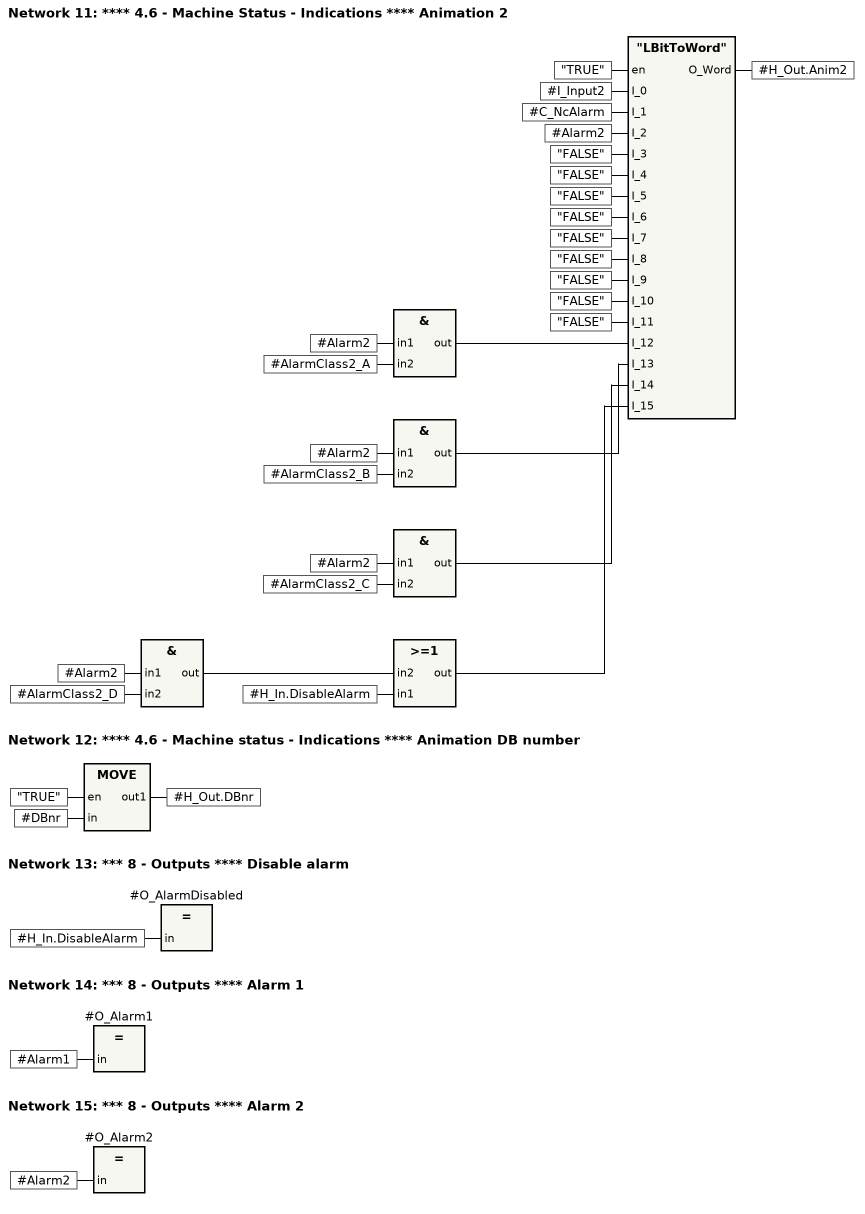
   IF "TRUE" THEN
       "LBitToWord"(I_0 := #I_Input2,
                    I_1 := #C_NcAlarm,
                    I_2 := #Alarm2,
                    I_3 := "FALSE",
                    I_4 := "FALSE",
                    I_5 := "FALSE",
                    I_6 := "FALSE",
                    I_7 := "FALSE",
                    I_8 := "FALSE",
                    I_9 := "FALSE",
                    I_10 := "FALSE",
                    I_11 := "FALSE",
                    I_12 := #Alarm2 AND #AlarmClass2_A,
                    I_13 := #Alarm2 AND #AlarmClass2_B,
                    I_14 := #Alarm2 AND #AlarmClass2_C,
                    I_15 := (#Alarm2 AND #AlarmClass2_D) OR #H_In.DisableAlarm,
                    O_Word => #H_Out.Anim2);
   END_IF;
END_REGION

REGION Network 12: **** 4.6 - Machine status - Indications **** Animation DB number
   IF "TRUE" THEN #H_Out.DBnr := #DBnr; END_IF;
END_REGION

REGION Network 13: *** 8 - Outputs **** Disable alarm
   // Alarm disabled from HMI
   #O_AlarmDisabled := #H_In.DisableAlarm;
END_REGION

REGION Network 14: *** 8 - Outputs **** Alarm 1
   // Output of the Alarm 1
   #O_Alarm1 := #Alarm1;
END_REGION

REGION Network 15: *** 8 - Outputs **** Alarm 2
   // Output of the Alarm 2
   #O_Alarm2 := #Alarm2;
END_REGION

REGION Network 16: **** 8 - Outputs **** Alarm AB Condition
   // Alarm AB condition
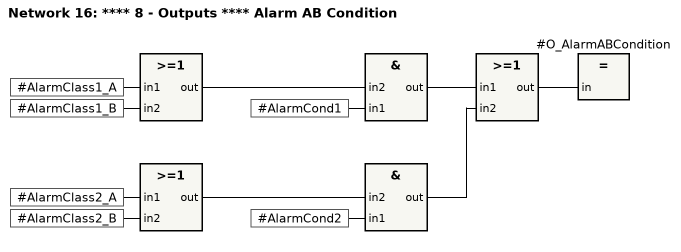
   #O_AlarmABCondition := ((#AlarmClass1_A OR #AlarmClass1_B) AND #AlarmCond1) OR ((#AlarmClass2_A OR #AlarmClass2_B) AND #AlarmCond2);
END_REGION
END_FUNCTION_BLOCK

FUNCTION_BLOCK "LPartDet"   // FB1610, FBD
TITLE = LPartDet
{ S7_Optimized_Access := 'FALSE' }
AUTHOR : VCC
FAMILY : ToolEqp
NAME : LPartDet
VERSION : 1.1
// ===============================================================================
// This module handles a partdetection with all his functions and alarms
// Functions are DetCheckOn, DetCheckOff and EnableAlarm
// Outputs are DetAlarm and DetOn signal
// ===============================================================================
// stored: AutoNumber false, IsIECCheckEnabled false, SetENOAutomatically False, UDAEnableTagReadback false
   VAR_INPUT
      I_SignalCheckOn { ExternalAccessible := 'False'; ExternalVisible := 'False'; ExternalWritable := 'False'} : Bool;   // Signal to check signal is on
      I_Signal { ExternalAccessible := 'False'; ExternalVisible := 'False'; ExternalWritable := 'False'} : Bool;   // Actual input from sensor
      I_SignalCheckOff { ExternalAccessible := 'False'; ExternalVisible := 'False'; ExternalWritable := 'False'} : Bool;   // Signal to check signal is off
      I_Simulate : Bool;   // Simulation mode
      I_AlarmClass { ExternalAccessible := 'False'; ExternalVisible := 'False'; ExternalWritable := 'False'} : Char;   // Alarm class -> A - B - C - D or E
      I_EnableAlarm { ExternalAccessible := 'False'; ExternalVisible := 'False'; ExternalWritable := 'False'} : Bool;   // Enable alarms
   END_VAR
   VAR_OUTPUT
      O_DetAlarm { ExternalAccessible := 'False'; ExternalVisible := 'False'; ExternalWritable := 'False'} : Bool;   // Detection alarm
      O_DetOn { ExternalAccessible := 'False'; ExternalVisible := 'False'; ExternalWritable := 'False'} : Bool;   // Detection signal to use in program
      H_IAnim { ExternalAccessible := 'False'; ExternalVisible := 'False'; ExternalWritable := 'False'} : Word;   // For animation of the icon
   END_VAR
   VAR DB_SPECIFIC
      H_Out : Struct   // HMI
         Anim : Word;   // HMI Animation of the object
         DBnr : Int;   // HMI Animation DB number
      END_STRUCT;
      DetCheckOnAlarm { ExternalAccessible := 'False'; ExternalVisible := 'False'; ExternalWritable := 'False'} : Bool;   // Detection is not on
      DetCheckOffAlarm { ExternalAccessible := 'False'; ExternalVisible := 'False'; ExternalWritable := 'False'} : Bool;   // Detection is not off
      DetOn { ExternalAccessible := 'False'; ExternalVisible := 'False'; ExternalWritable := 'False'} : Bool;   // Detection on
      DetAlarm { ExternalAccessible := 'False'; ExternalVisible := 'False'; ExternalWritable := 'False'} : Bool;   // Detection alarm
      AlarmClass_A { ExternalAccessible := 'False'; ExternalVisible := 'False'; ExternalWritable := 'False'} : Bool;   // The alarm is from alarm class A
      AlarmClass_B { ExternalAccessible := 'False'; ExternalVisible := 'False'; ExternalWritable := 'False'} : Bool;   // The alarm is from alarm class B
      AlarmClass_C { ExternalAccessible := 'False'; ExternalVisible := 'False'; ExternalWritable := 'False'} : Bool;   // The alarm is from alarm class C
      AlarmClass_D { ExternalAccessible := 'False'; ExternalVisible := 'False'; ExternalWritable := 'False'} : Bool;   // The alarm is from alarm class D
      AlarmClass_E { ExternalAccessible := 'False'; ExternalVisible := 'False'; ExternalWritable := 'False'} : Bool;   // The alarm is from alarm class E
      DBnr { ExternalAccessible := 'False'; ExternalVisible := 'False'; ExternalWritable := 'False'} : Int;   // HMI DB number
   END_VAR
BEGIN

NETWORK
TITLE = **** 1 - Inputs **** DB number
// DB number
      L     DINO;
      T     #DBnr;

NETWORK
TITLE = **** 1 - Inputs **** Alarm class
// Alarm class
// Alarm class = E
      L     #I_AlarmClass;
      L     'E';
      ==I;
      =     #AlarmClass_E;

// Alarm class = D
      L     #I_AlarmClass;
      L     'D';
      ==I;
      =     #AlarmClass_D;

// Alarm class = C
      L     #I_AlarmClass;
      L     'C';
      ==I;
      =     #AlarmClass_C;

// Alarm class = B
      L     #I_AlarmClass;
      L     'B';
      ==I;
      =     #AlarmClass_B;

// Alarm class = A
      AN    #AlarmClass_B;
      AN    #AlarmClass_C;
      AN    #AlarmClass_D;
      AN    #AlarmClass_E;
      =     #AlarmClass_A;


REGION Network 3: **** 2.2 - Alarms - Alarm generation **** Creating alarm for active detection
   // Creating alarm for active detection
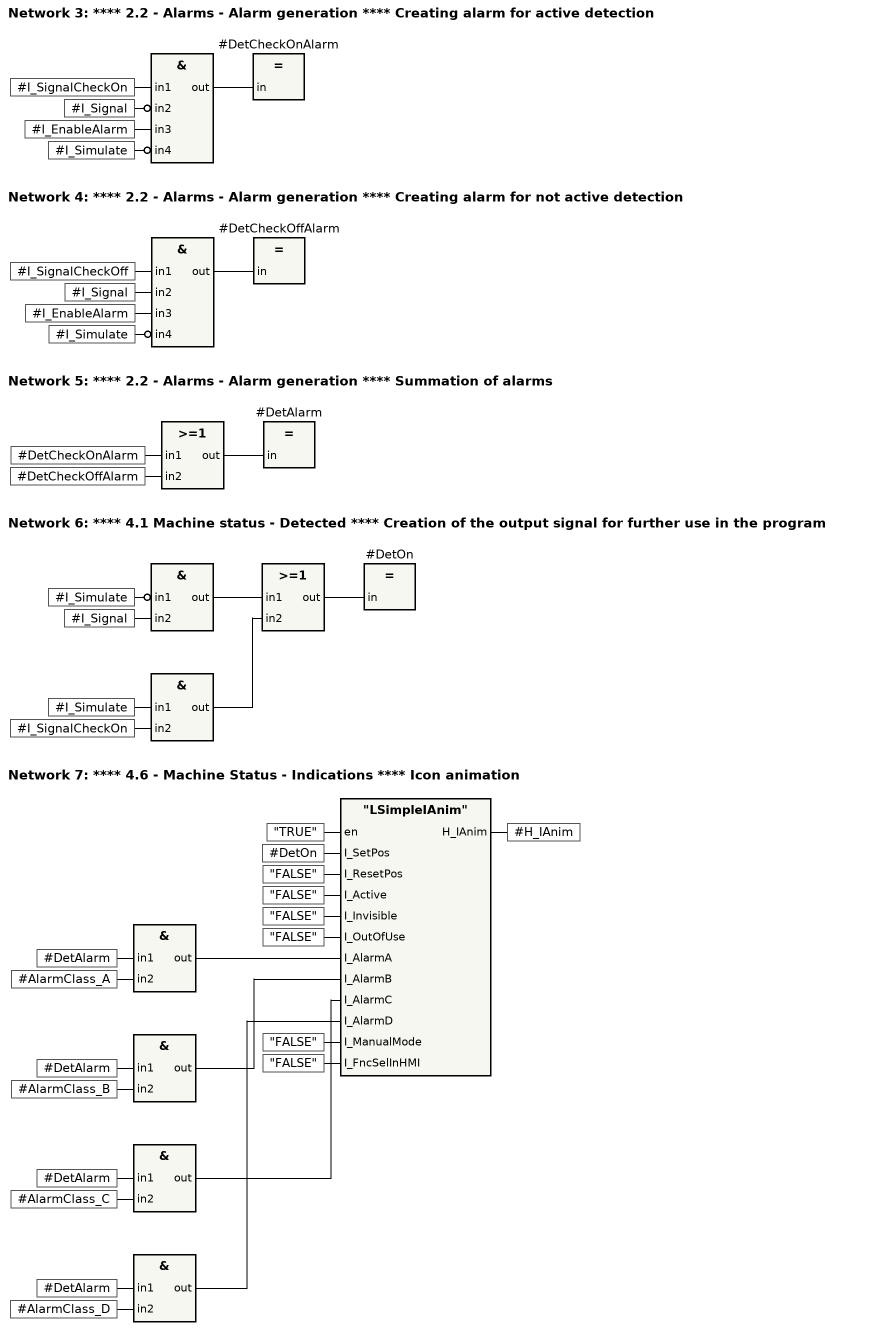
   #DetCheckOnAlarm := #I_SignalCheckOn AND NOT #I_Signal AND #I_EnableAlarm AND NOT #I_Simulate;
END_REGION

REGION Network 4: **** 2.2 - Alarms - Alarm generation **** Creating alarm for not active detection
   // Creating alarm for not active detection
   #DetCheckOffAlarm := #I_SignalCheckOff AND #I_Signal AND #I_EnableAlarm AND NOT #I_Simulate;
END_REGION

REGION Network 5: **** 2.2 - Alarms - Alarm generation **** Summation of alarms
   // Summation of alarms
   #DetAlarm := #DetCheckOnAlarm OR #DetCheckOffAlarm;
END_REGION

REGION Network 6: **** 4.1 Machine status - Detected **** Creation of the output signal for further use in the program
   // Creation of the output signal for further use in the program
   #DetOn := (NOT #I_Simulate AND #I_Signal) OR (#I_Simulate AND #I_SignalCheckOn);
END_REGION

REGION Network 7: **** 4.6 - Machine Status - Indications **** Icon animation
   // Icon animation
   IF "TRUE" THEN
       "LSimpleIAnim"(I_SetPos := #DetOn,
                      I_ResetPos := "FALSE",
                      I_Active := "FALSE",
                      I_Invisible := "FALSE",
                      I_OutOfUse := "FALSE",
                      I_AlarmA := #DetAlarm AND #AlarmClass_A,
                      I_AlarmB := #DetAlarm AND #AlarmClass_B,
                      I_AlarmC := #DetAlarm AND #AlarmClass_C,
                      I_AlarmD := #DetAlarm AND #AlarmClass_D,
                      I_ManualMode := "FALSE",
                      I_FncSelInHMI := "FALSE",
                      H_IAnim => #H_IAnim);
   END_IF;
END_REGION

REGION Network 8: **** 4.6 - Machine Status - Indications **** Animation
   // Animation
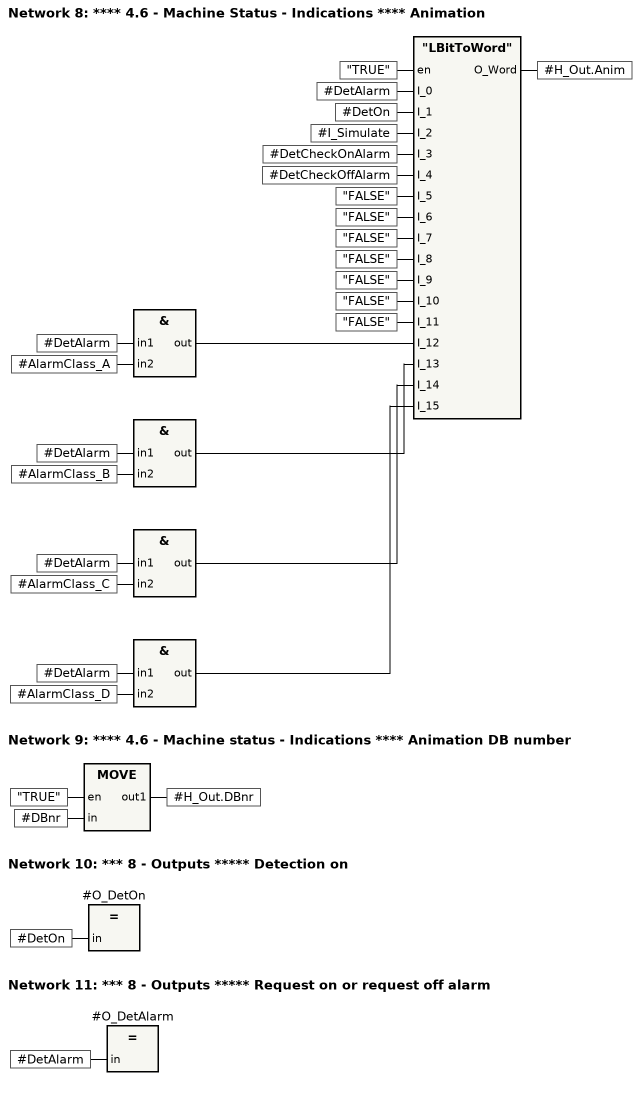
   IF "TRUE" THEN
       "LBitToWord"(I_0 := #DetAlarm,
                    I_1 := #DetOn,
                    I_2 := #I_Simulate,
                    I_3 := #DetCheckOnAlarm,
                    I_4 := #DetCheckOffAlarm,
                    I_5 := "FALSE",
                    I_6 := "FALSE",
                    I_7 := "FALSE",
                    I_8 := "FALSE",
                    I_9 := "FALSE",
                    I_10 := "FALSE",
                    I_11 := "FALSE",
                    I_12 := #DetAlarm AND #AlarmClass_A,
                    I_13 := #DetAlarm AND #AlarmClass_B,
                    I_14 := #DetAlarm AND #AlarmClass_C,
                    I_15 := #DetAlarm AND #AlarmClass_D,
                    O_Word => #H_Out.Anim);
   END_IF;
END_REGION

REGION Network 9: **** 4.6 - Machine status - Indications **** Animation DB number
   // Animation DB number
   IF "TRUE" THEN #H_Out.DBnr := #DBnr; END_IF;
END_REGION

REGION Network 10: *** 8 - Outputs ***** Detection on
   // Detection on
   #O_DetOn := #DetOn;
END_REGION

REGION Network 11: *** 8 - Outputs ***** Request on or request off alarm
   // Request on or request off alarm
   #O_DetAlarm := #DetAlarm;
END_REGION
END_FUNCTION_BLOCK

FUNCTION_BLOCK "LPartSensor"   // FB1614, FBD
TITLE = LPartDet
{ S7_Optimized_Access := 'FALSE' }
AUTHOR : VCC
FAMILY : ToolEqp
NAME : LPartSen
VERSION : 1.0
// ===============================================================================
// This module handles a partdetection with all his functions and alarms
// Functions are DetCheckOn, DetCheckOff and EnableAlarm
// Outputs are DetAlarm and DetOn signal
// ===============================================================================
// stored: AutoNumber false, IsIECCheckEnabled false, SetENOAutomatically False, UDAEnableTagReadback false
   VAR_INPUT
      I_SignalCheckOn { ExternalAccessible := 'False'; ExternalVisible := 'False'; ExternalWritable := 'False'} : Bool;   // Signal to check signal is on
      I_Signal { ExternalAccessible := 'False'; ExternalVisible := 'False'; ExternalWritable := 'False'} : Bool;   // Actual input from sensor
      I_SignalCheckOff { ExternalAccessible := 'False'; ExternalVisible := 'False'; ExternalWritable := 'False'} : Bool;   // Signal to check signal is off
      I_Simulate : Bool;   // Simulation mode
      I_AlarmClass { ExternalAccessible := 'False'; ExternalVisible := 'False'; ExternalWritable := 'False'} : Char;   // Alarm class -> A - B - C - D or E
      I_EnableAlarm { ExternalAccessible := 'False'; ExternalVisible := 'False'; ExternalWritable := 'False'} : Bool;   // Enable alarms
      I_AlarmResetPB { ExternalAccessible := 'False'; ExternalVisible := 'False'; ExternalWritable := 'False'} : Bool;   // Alarm reset pushbutton is activated
   END_VAR
   VAR_OUTPUT
      O_DetOn { ExternalAccessible := 'False'; ExternalVisible := 'False'; ExternalWritable := 'False'} : Bool;   // Detection signal to use in program
      O_DetAlmReqOn { ExternalAccessible := 'False'; ExternalVisible := 'False'; ExternalWritable := 'False'} : Bool;   // Request on alarm
      O_DetAlmReqOff { ExternalAccessible := 'False'; ExternalVisible := 'False'; ExternalWritable := 'False'} : Bool;   // Request off alarm
      O_DetSumAlm { ExternalAccessible := 'False'; ExternalVisible := 'False'; ExternalWritable := 'False'} : Bool;   // Request on or request off signal active
      O_AlarmABCondition { ExternalAccessible := 'False'; ExternalVisible := 'False'; ExternalWritable := 'False'} : Bool;   // Alarm AB condition
      H_IAnim { ExternalAccessible := 'False'; ExternalVisible := 'False'; ExternalWritable := 'False'} : Word;   // For animation of the icon
   END_VAR
   VAR DB_SPECIFIC
      H_Out : Struct   // HMI
         Anim : Word;   // HMI Animation of the object
         DBnr : Int;   // HMI Animation DB number
      END_STRUCT;
      DetCheckOnAlarm { ExternalAccessible := 'False'; ExternalVisible := 'False'; ExternalWritable := 'False'} : Bool;   // Detection is not on
      DetCheckOffAlarm { ExternalAccessible := 'False'; ExternalVisible := 'False'; ExternalWritable := 'False'} : Bool;   // Detection is not off
      DetOn { ExternalAccessible := 'False'; ExternalVisible := 'False'; ExternalWritable := 'False'} : Bool;   // Detection on
      DetAlarm { ExternalAccessible := 'False'; ExternalVisible := 'False'; ExternalWritable := 'False'} : Bool;   // Detection alarm
      AlarmCondReqOn { ExternalAccessible := 'False'; ExternalVisible := 'False'; ExternalWritable := 'False'} : Bool;   // Alarm condition
      AlarmCondReqOff { ExternalAccessible := 'False'; ExternalVisible := 'False'; ExternalWritable := 'False'} : Bool;   // Alarm condition
      AlarmClass_A { ExternalAccessible := 'False'; ExternalVisible := 'False'; ExternalWritable := 'False'} : Bool;   // The alarm is from alarm class A
      AlarmClass_B { ExternalAccessible := 'False'; ExternalVisible := 'False'; ExternalWritable := 'False'} : Bool;   // The alarm is from alarm class B
      AlarmClass_C { ExternalAccessible := 'False'; ExternalVisible := 'False'; ExternalWritable := 'False'} : Bool;   // The alarm is from alarm class C
      AlarmClass_D { ExternalAccessible := 'False'; ExternalVisible := 'False'; ExternalWritable := 'False'} : Bool;   // The alarm is from alarm class D
      AlarmClass_E { ExternalAccessible := 'False'; ExternalVisible := 'False'; ExternalWritable := 'False'} : Bool;   // The alarm is from alarm class E
      DBnr { ExternalAccessible := 'False'; ExternalVisible := 'False'; ExternalWritable := 'False'} : Int;   // HMI DB number
   END_VAR
BEGIN

NETWORK
TITLE = **** 1 - Inputs **** DB number
// DB number
      L     DINO;
      T     #DBnr;

NETWORK
TITLE = **** 1 - Inputs **** Alarm class
// Alarm class
// Alarm class = E
      L     #I_AlarmClass;
      L     'E';
      ==I;
      =     #AlarmClass_E;

// Alarm class = D
      L     #I_AlarmClass;
      L     'D';
      ==I;
      =     #AlarmClass_D;

// Alarm class = C
      L     #I_AlarmClass;
      L     'C';
      ==I;
      =     #AlarmClass_C;

// Alarm class = B
      L     #I_AlarmClass;
      L     'B';
      ==I;
      =     #AlarmClass_B;

// Alarm class = A
      AN    #AlarmClass_B;
      AN    #AlarmClass_C;
      AN    #AlarmClass_D;
      AN    #AlarmClass_E;
      =     #AlarmClass_A;


REGION Network 3: **** 2.2 - Alarms - Alarm generation **** Condition alarm for active detection
   // Condition alarm for active detection
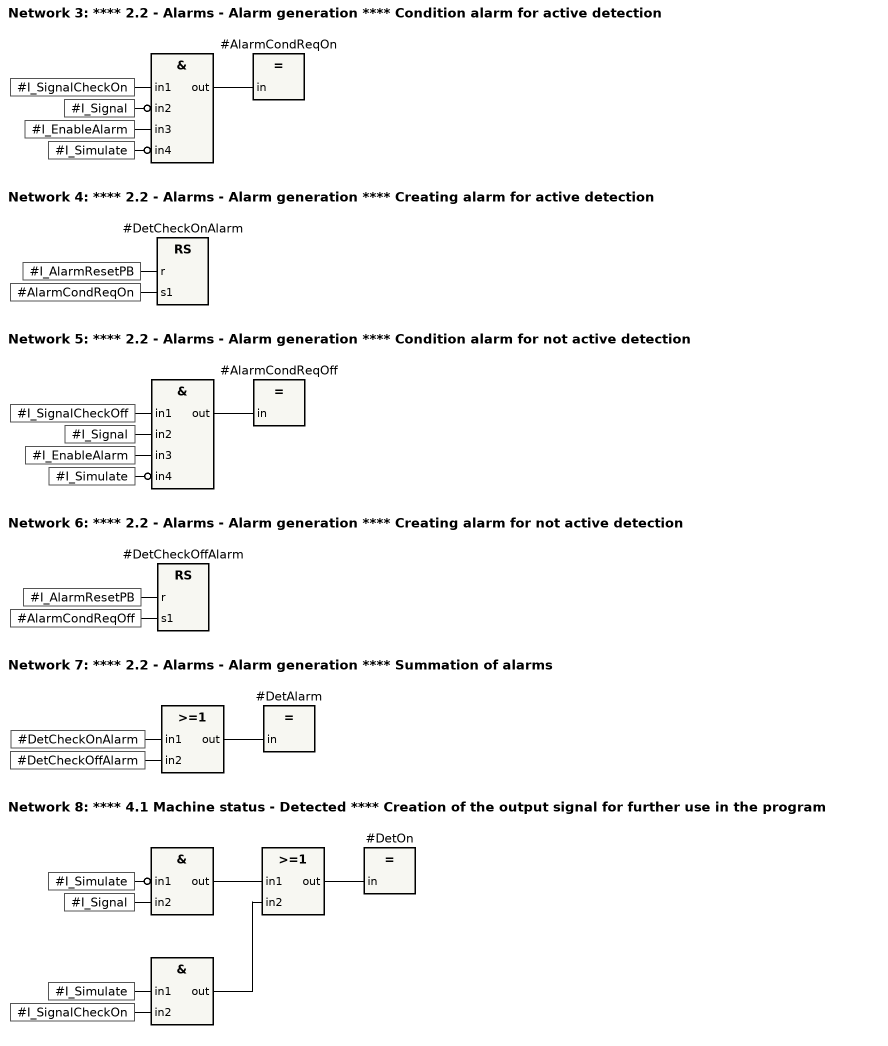
   #AlarmCondReqOn := #I_SignalCheckOn AND NOT #I_Signal AND #I_EnableAlarm AND NOT #I_Simulate;
END_REGION

REGION Network 4: **** 2.2 - Alarms - Alarm generation **** Creating alarm for active detection
   // Creating alarm for active detection
   IF #I_AlarmResetPB THEN
       #DetCheckOnAlarm := FALSE;   // RS flip-flop
   END_IF;
   IF #AlarmCondReqOn THEN #DetCheckOnAlarm := TRUE; END_IF;
END_REGION

REGION Network 5: **** 2.2 - Alarms - Alarm generation **** Condition alarm for not active detection
   // Condition alarm for not active detection
   #AlarmCondReqOff := #I_SignalCheckOff AND #I_Signal AND #I_EnableAlarm AND NOT #I_Simulate;
END_REGION

REGION Network 6: **** 2.2 - Alarms - Alarm generation **** Creating alarm for not active detection
   // Creating alarm for not active detection
   IF #I_AlarmResetPB THEN
       #DetCheckOffAlarm := FALSE;   // RS flip-flop
   END_IF;
   IF #AlarmCondReqOff THEN #DetCheckOffAlarm := TRUE; END_IF;
END_REGION

REGION Network 7: **** 2.2 - Alarms - Alarm generation **** Summation of alarms
   // Summation of alarms
   #DetAlarm := #DetCheckOnAlarm OR #DetCheckOffAlarm;
END_REGION

REGION Network 8: **** 4.1 Machine status - Detected **** Creation of the output signal for further use in the program
   // Creation of the output signal for further use in the program
   #DetOn := (NOT #I_Simulate AND #I_Signal) OR (#I_Simulate AND #I_SignalCheckOn);
END_REGION

REGION Network 9: **** 4.6 - Machine Status - Indications **** Icon animation
   // Icon animation
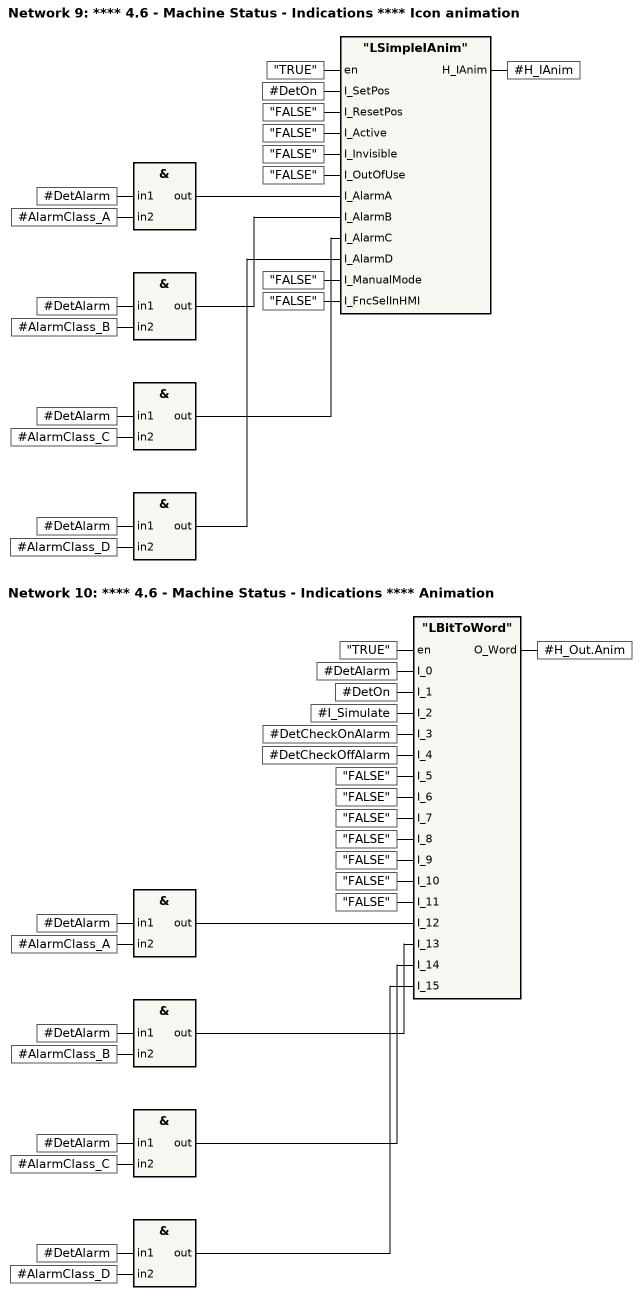
   IF "TRUE" THEN
       "LSimpleIAnim"(I_SetPos := #DetOn,
                      I_ResetPos := "FALSE",
                      I_Active := "FALSE",
                      I_Invisible := "FALSE",
                      I_OutOfUse := "FALSE",
                      I_AlarmA := #DetAlarm AND #AlarmClass_A,
                      I_AlarmB := #DetAlarm AND #AlarmClass_B,
                      I_AlarmC := #DetAlarm AND #AlarmClass_C,
                      I_AlarmD := #DetAlarm AND #AlarmClass_D,
                      I_ManualMode := "FALSE",
                      I_FncSelInHMI := "FALSE",
                      H_IAnim => #H_IAnim);
   END_IF;
END_REGION

REGION Network 10: **** 4.6 - Machine Status - Indications **** Animation
   // Animation
   IF "TRUE" THEN
       "LBitToWord"(I_0 := #DetAlarm,
                    I_1 := #DetOn,
                    I_2 := #I_Simulate,
                    I_3 := #DetCheckOnAlarm,
                    I_4 := #DetCheckOffAlarm,
                    I_5 := "FALSE",
                    I_6 := "FALSE",
                    I_7 := "FALSE",
                    I_8 := "FALSE",
                    I_9 := "FALSE",
                    I_10 := "FALSE",
                    I_11 := "FALSE",
                    I_12 := #DetAlarm AND #AlarmClass_A,
                    I_13 := #DetAlarm AND #AlarmClass_B,
                    I_14 := #DetAlarm AND #AlarmClass_C,
                    I_15 := #DetAlarm AND #AlarmClass_D,
                    O_Word => #H_Out.Anim);
   END_IF;
END_REGION

REGION Network 11: **** 4.6 - Machine status - Indications **** Animation DB number
   // Animation DB number
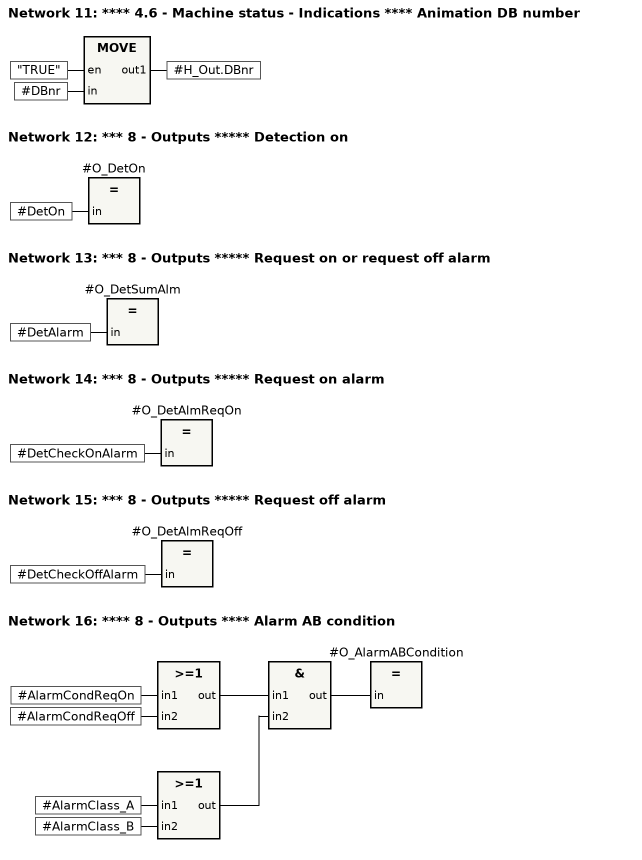
   IF "TRUE" THEN #H_Out.DBnr := #DBnr; END_IF;
END_REGION

REGION Network 12: *** 8 - Outputs ***** Detection on
   // Detection on
   #O_DetOn := #DetOn;
END_REGION

REGION Network 13: *** 8 - Outputs ***** Request on or request off alarm
   // Request on or request off alarm
   #O_DetSumAlm := #DetAlarm;
END_REGION

REGION Network 14: *** 8 - Outputs ***** Request on alarm
   // Request on alarm
   #O_DetAlmReqOn := #DetCheckOnAlarm;
END_REGION

REGION Network 15: *** 8 - Outputs ***** Request off alarm
   // Request off alarm
   #O_DetAlmReqOff := #DetCheckOffAlarm;
END_REGION

REGION Network 16: **** 8 - Outputs **** Alarm AB condition
   // Alarm AB condition
   #O_AlarmABCondition := (#AlarmCondReqOn OR #AlarmCondReqOff) AND (#AlarmClass_A OR #AlarmClass_B);
END_REGION
END_FUNCTION_BLOCK

FUNCTION_BLOCK "LProcAnInput6Lim"   // FB1700, FBD
TITLE = LAnInput6Lim / LProcAnInput6Lim
{ S7_Optimized_Access := 'FALSE' }
AUTHOR : VCC
FAMILY : ProcEqp
NAME : AnInput
VERSION : 1.0
// ================================================================================
// This module is used to read an analogue Input value and scale it. 
// It also gives the possibility to define 6 limits (High High High, High High, 
// High, Low, Low Low and Low Low Low level) and to create 6 alarms for these 
// limits. 
// ================================================================================
// stored: AutoNumber false, IsIECCheckEnabled false, SetENOAutomatically False, UDAEnableTagReadback false
   VAR_INPUT
      I_AnInput { ExternalAccessible := 'False'; ExternalVisible := 'False'; ExternalWritable := 'False'} : Int;   // Analogue Input Value
      I_AnInput_Bipolar { ExternalAccessible := 'False'; ExternalVisible := 'False'; ExternalWritable := 'False'} : Bool;   // TRUE if Analogue Input Bipolar
      I_EnHHHAlarm { ExternalAccessible := 'False'; ExternalVisible := 'False'; ExternalWritable := 'False'} : Bool;   // Enable HHH Limit Alarm
      I_ResHHHAlarm { ExternalAccessible := 'False'; ExternalVisible := 'False'; ExternalWritable := 'False'} : Bool;   // Reset HHH Limit Alarm
      I_EnHHAlarm { ExternalAccessible := 'False'; ExternalVisible := 'False'; ExternalWritable := 'False'} : Bool;   // Enable HH Limit Alarm
      I_ResHHAlarm { ExternalAccessible := 'False'; ExternalVisible := 'False'; ExternalWritable := 'False'} : Bool;   // Reset HH Limit Alarm
      I_EnHAlarm { ExternalAccessible := 'False'; ExternalVisible := 'False'; ExternalWritable := 'False'} : Bool;   // Enable H Limit Alarm
      I_ResHAlarm { ExternalAccessible := 'False'; ExternalVisible := 'False'; ExternalWritable := 'False'} : Bool;   // Reset H Limit Alarm
      I_EnLAlarm { ExternalAccessible := 'False'; ExternalVisible := 'False'; ExternalWritable := 'False'} : Bool;   // Enable L Limit Alarm
      I_ResLAlarm { ExternalAccessible := 'False'; ExternalVisible := 'False'; ExternalWritable := 'False'} : Bool;   // Reset L Limit Alarm
      I_EnLLAlarm { ExternalAccessible := 'False'; ExternalVisible := 'False'; ExternalWritable := 'False'} : Bool;   // Enable LL Limit Alarm
      I_ResLLAlarm { ExternalAccessible := 'False'; ExternalVisible := 'False'; ExternalWritable := 'False'} : Bool;   // Reset LL Limit Alarm
      I_EnLLLAlarm { ExternalAccessible := 'False'; ExternalVisible := 'False'; ExternalWritable := 'False'} : Bool;   // Enable LLL Limit Alarm
      I_ResLLLAlarm { ExternalAccessible := 'False'; ExternalVisible := 'False'; ExternalWritable := 'False'} : Bool;   // Reset LLL Limit Alarm
      I_AlarmResetPB { ExternalAccessible := 'False'; ExternalVisible := 'False'; ExternalWritable := 'False'} : Bool;   // Alarm reset PB
   END_VAR
   VAR_OUTPUT
      O_SensorAlarm { ExternalAccessible := 'False'; ExternalVisible := 'False'; ExternalWritable := 'False'} : Bool;   // Sensor out of range
      O_HHHAlarm { ExternalAccessible := 'False'; ExternalVisible := 'False'; ExternalWritable := 'False'} : Bool;   // HHH Limit Alarm
      O_HHAlarm { ExternalAccessible := 'False'; ExternalVisible := 'False'; ExternalWritable := 'False'} : Bool;   // HH Limit Alarm
      O_HAlarm { ExternalAccessible := 'False'; ExternalVisible := 'False'; ExternalWritable := 'False'} : Bool;   // H Limit Alarm
      O_LAlarm { ExternalAccessible := 'False'; ExternalVisible := 'False'; ExternalWritable := 'False'} : Bool;   // L Limit Alarm
      O_LLAlarm { ExternalAccessible := 'False'; ExternalVisible := 'False'; ExternalWritable := 'False'} : Bool;   // LL Limit Alarm
      O_LLLAlarm { ExternalAccessible := 'False'; ExternalVisible := 'False'; ExternalWritable := 'False'} : Bool;   // LLL Limit Alarm
      O_AnInputScaled : Real;   // Analogue Input value after scaling
      O_AlarmABCondition { ExternalAccessible := 'False'; ExternalVisible := 'False'; ExternalWritable := 'False'} : Bool;   // Alarm AB condition
      O_HHHReached { ExternalAccessible := 'False'; ExternalVisible := 'False'; ExternalWritable := 'False'} : Bool;   // High High High Limit Reached
      O_HHReached { ExternalAccessible := 'False'; ExternalVisible := 'False'; ExternalWritable := 'False'} : Bool;   // High High Limit Reached
      O_HReached { ExternalAccessible := 'False'; ExternalVisible := 'False'; ExternalWritable := 'False'} : Bool;   // High Limit Reached
      O_LReached { ExternalAccessible := 'False'; ExternalVisible := 'False'; ExternalWritable := 'False'} : Bool;   // Low Limit Reached
      O_LLReached { ExternalAccessible := 'False'; ExternalVisible := 'False'; ExternalWritable := 'False'} : Bool;   // Low Low Limit Reached
      O_LLLReached { ExternalAccessible := 'False'; ExternalVisible := 'False'; ExternalWritable := 'False'} : Bool;   // Low Low Low Limit Reached
      H_IAnim { ExternalAccessible := 'False'; ExternalVisible := 'False'; ExternalWritable := 'False'} : Word;   // HMI Animation of the icon
   END_VAR
   VAR DB_SPECIFIC
      H_In : Struct   // HMI
         AnInput_HighLimit : Real;   // From HMI : High Limit For Scaling Analogue Input
         AnInput_LowLimit : Real;   // From HMI : Low Limit For Scaling Analogue Input
         HHysteresis : Real;   // From HMI : Hysteresis value for High Limits
         LHysteresis : Real;   // From HMI : Hysteresis value for Low Limits
         HHHLimitValue : Real;   // From HMI : High High High Limit Value
         HHLimitValue : Real;   // From HMI : High High Limit Value
         HLimitValue : Real;   // From HMI : High Limit Value
         LLimitValue : Real;   // From HMI : Low Limit Value
         LLLimitValue : Real;   // From HMI : Low Low Limit Value
         LLLLimitValue : Real;   // From HMI : Low Low Low Limit Value
         TimeDelay : DInt;   // From HMI : Time delay for limits
         Forcing : Bool;   // From HMI : True if forced value must be used
         ForcedAnInput : Real;   // From HMI : Forced Analogue Input Value
      END_STRUCT;
      H_Out : Struct   // HMI
         Anim : Word;   // HMI Animation of the object
         DBnr : Int;   // HMI Animation DB number
      END_STRUCT;
   END_VAR
   VAR
      HHHLimitTimer { ExternalAccessible := 'False'; ExternalVisible := 'False'; ExternalWritable := 'False'; S7_SetPoint := 'True'} : "LTimer";   // Timer HHH Limit
      HHLimitTimer { ExternalAccessible := 'False'; ExternalVisible := 'False'; ExternalWritable := 'False'; S7_SetPoint := 'True'} : "LTimer";   // Timer HH Limit
      HLimitTimer { ExternalAccessible := 'False'; ExternalVisible := 'False'; ExternalWritable := 'False'; S7_SetPoint := 'True'} : "LTimer";   // Timer H Limit
      LLimitTimer { ExternalAccessible := 'False'; ExternalVisible := 'False'; ExternalWritable := 'False'; S7_SetPoint := 'True'} : "LTimer";   // Timer L Limit
      LLLimitTimer { ExternalAccessible := 'False'; ExternalVisible := 'False'; ExternalWritable := 'False'; S7_SetPoint := 'True'} : "LTimer";   // Timer LL Limit
      LLLLimitTimer { ExternalAccessible := 'False'; ExternalVisible := 'False'; ExternalWritable := 'False'; S7_SetPoint := 'True'} : "LTimer";   // Timer LLL Limit
   END_VAR
   VAR DB_SPECIFIC
      AnInputScaled { ExternalAccessible := 'False'; ExternalVisible := 'False'; ExternalWritable := 'False'} : Real;   // Analogue Input value after scaling
      HHHTempSR { ExternalAccessible := 'False'; ExternalVisible := 'False'; ExternalWritable := 'False'} : Bool;   // Temp variable for SET/RESET
      HHTempSR { ExternalAccessible := 'False'; ExternalVisible := 'False'; ExternalWritable := 'False'} : Bool;   // Temp variable for SET/RESET
      HTempSR { ExternalAccessible := 'False'; ExternalVisible := 'False'; ExternalWritable := 'False'} : Bool;   // Temp variable for SET/RESET
      LTempSR { ExternalAccessible := 'False'; ExternalVisible := 'False'; ExternalWritable := 'False'} : Bool;   // Temp variable for SET/RESET
      LLTempSR { ExternalAccessible := 'False'; ExternalVisible := 'False'; ExternalWritable := 'False'} : Bool;   // Temp variable for SET/RESET
      LLLTempSR { ExternalAccessible := 'False'; ExternalVisible := 'False'; ExternalWritable := 'False'} : Bool;   // Temp variable for SET/RESET
      Scale_status { ExternalAccessible := 'False'; ExternalVisible := 'False'; ExternalWritable := 'False'} : Word;   // Status word for scaling operation
      HHHlimitHyst { ExternalAccessible := 'False'; ExternalVisible := 'False'; ExternalWritable := 'False'} : Real;   // HHH Limit with Hysteresis
      HHlimitHyst { ExternalAccessible := 'False'; ExternalVisible := 'False'; ExternalWritable := 'False'} : Real;   // HH Limit with Hysteresis
      HlimitHyst { ExternalAccessible := 'False'; ExternalVisible := 'False'; ExternalWritable := 'False'} : Real;   // H Limit with Hysteresis
      LlimitHyst { ExternalAccessible := 'False'; ExternalVisible := 'False'; ExternalWritable := 'False'} : Real;   // L Limit with Hysteresis
      LLlimitHyst { ExternalAccessible := 'False'; ExternalVisible := 'False'; ExternalWritable := 'False'} : Real;   // LL Limit with Hysteresis
      LLLlimitHyst { ExternalAccessible := 'False'; ExternalVisible := 'False'; ExternalWritable := 'False'} : Real;   // LLL Limit with Hysteresis
      HHHReached { ExternalAccessible := 'False'; ExternalVisible := 'False'; ExternalWritable := 'False'} : Bool;   // Temp variable HHH Limit Reached
      HHReached { ExternalAccessible := 'False'; ExternalVisible := 'False'; ExternalWritable := 'False'} : Bool;   // Temp variable HH Limit Reached
      HReached { ExternalAccessible := 'False'; ExternalVisible := 'False'; ExternalWritable := 'False'} : Bool;   // Temp variable H Limit Reached
      LReached { ExternalAccessible := 'False'; ExternalVisible := 'False'; ExternalWritable := 'False'} : Bool;   // Temp variable L Limit Reached
      LLReached { ExternalAccessible := 'False'; ExternalVisible := 'False'; ExternalWritable := 'False'} : Bool;   // Temp variable LL Limit Reached
      LLLReached { ExternalAccessible := 'False'; ExternalVisible := 'False'; ExternalWritable := 'False'} : Bool;   // Temp variable LLL Limit Reached
      HHHAlarmAlmCond { ExternalAccessible := 'False'; ExternalVisible := 'False'; ExternalWritable := 'False'} : Bool;   // HHHAlarm alarm condition
      HHAlarmAlmCond { ExternalAccessible := 'False'; ExternalVisible := 'False'; ExternalWritable := 'False'} : Bool;   // HHAlarm alarm condition
      HAlarmAlmCond { ExternalAccessible := 'False'; ExternalVisible := 'False'; ExternalWritable := 'False'} : Bool;   // HAlarm alarm condition
      LAlarmAlmCond { ExternalAccessible := 'False'; ExternalVisible := 'False'; ExternalWritable := 'False'} : Bool;   // LAlarm alarm condition
      LLAlarmAlmCond { ExternalAccessible := 'False'; ExternalVisible := 'False'; ExternalWritable := 'False'} : Bool;   // LLAlarm alarm condition
      LLLAlarmAlmCond { ExternalAccessible := 'False'; ExternalVisible := 'False'; ExternalWritable := 'False'} : Bool;   // LLLAlarm alarm condition
      HHHAlarm { ExternalAccessible := 'False'; ExternalVisible := 'False'; ExternalWritable := 'False'} : Bool;   // HHH Limit Alarm
      HHAlarm { ExternalAccessible := 'False'; ExternalVisible := 'False'; ExternalWritable := 'False'} : Bool;   // HH Limit Alarm
      HAlarm { ExternalAccessible := 'False'; ExternalVisible := 'False'; ExternalWritable := 'False'} : Bool;   // H Limit Alarm
      LAlarm { ExternalAccessible := 'False'; ExternalVisible := 'False'; ExternalWritable := 'False'} : Bool;   // L Limit Alarm
      LLAlarm { ExternalAccessible := 'False'; ExternalVisible := 'False'; ExternalWritable := 'False'} : Bool;   // LL Limit Alarm
      LLLAlarm { ExternalAccessible := 'False'; ExternalVisible := 'False'; ExternalWritable := 'False'} : Bool;   // LLL Limit Alarm
      SensorAlarm { ExternalAccessible := 'False'; ExternalVisible := 'False'; ExternalWritable := 'False'} : Bool;   // Sensor out of range
      SensorAlmCond { ExternalAccessible := 'False'; ExternalVisible := 'False'; ExternalWritable := 'False'} : Bool;   // Sensor alarm condition
      ScaleRetValue { ExternalAccessible := 'False'; ExternalVisible := 'False'; ExternalWritable := 'False'} : Int;   // Scale return value
      AnInputTmp { ExternalAccessible := 'False'; ExternalVisible := 'False'; ExternalWritable := 'False'} : Real;   // Analog input temporary
      DBnr { ExternalAccessible := 'False'; ExternalVisible := 'False'; ExternalWritable := 'False'} : Int;   // HMI DB number
   END_VAR
   VAR
      HHH_Alarm { ExternalAccessible := 'False'; ExternalVisible := 'False'; ExternalWritable := 'False'; S7_SetPoint := 'True'} : "LProc1AlarmMultiIn";
      HH_Alarm { ExternalAccessible := 'False'; ExternalVisible := 'False'; ExternalWritable := 'False'; S7_SetPoint := 'True'} : "LProc1AlarmMultiIn";
      H_Alarm { ExternalAccessible := 'False'; ExternalVisible := 'False'; ExternalWritable := 'False'; S7_SetPoint := 'True'} : "LProc1AlarmMultiIn";
      L_Alarm { ExternalAccessible := 'False'; ExternalVisible := 'False'; ExternalWritable := 'False'; S7_SetPoint := 'True'} : "LProc1AlarmMultiIn";
      LL_Alarm { ExternalAccessible := 'False'; ExternalVisible := 'False'; ExternalWritable := 'False'; S7_SetPoint := 'True'} : "LProc1AlarmMultiIn";
      LLL_Alarm { ExternalAccessible := 'False'; ExternalVisible := 'False'; ExternalWritable := 'False'; S7_SetPoint := 'True'} : "LProc1AlarmMultiIn";
      SensorAlm { ExternalAccessible := 'False'; ExternalVisible := 'False'; ExternalWritable := 'False'; S7_SetPoint := 'True'} : "LProc1AlarmMultiIn";
   END_VAR
BEGIN

NETWORK
TITLE = **** 1 - Inputs **** DB number
// DB number
      L     DINO;
      T     #DBnr;

REGION Network 2: **** 2.2 - Alarms - Alarm generation **** Alarm High High High Limit
   // Alarm High High High Limit
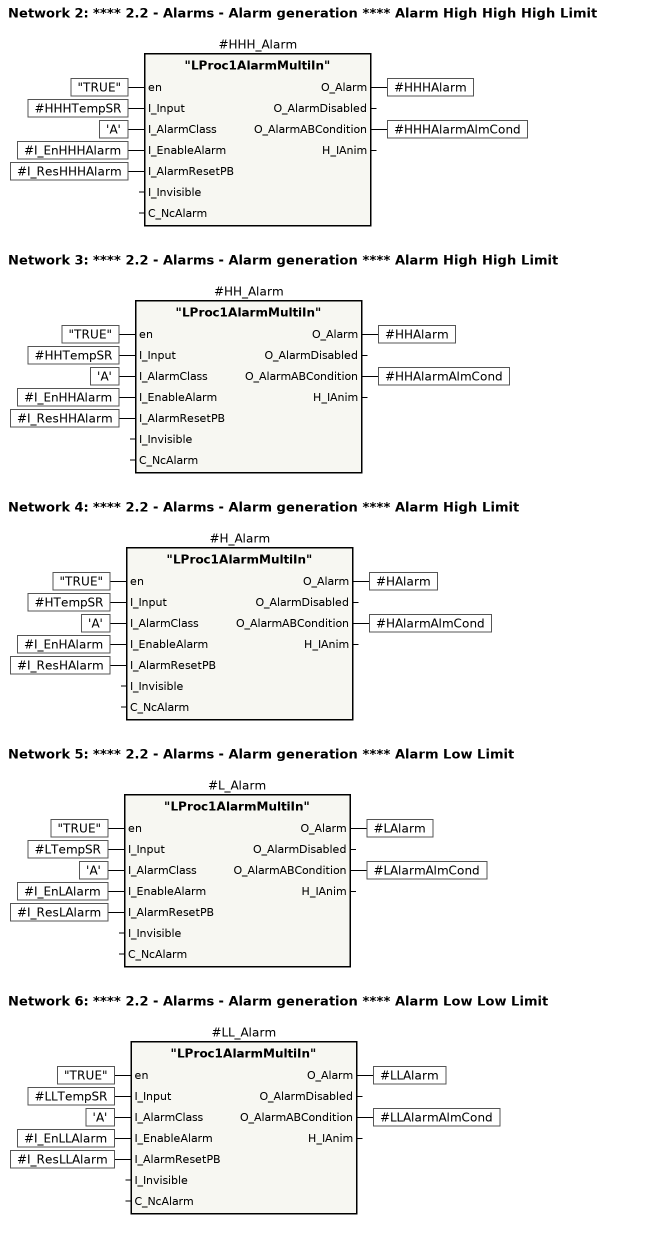
   IF "TRUE" THEN
       #HHH_Alarm(I_Input := #HHHTempSR,   // "LProc1AlarmMultiIn"
                  I_AlarmClass := 'A',
                  I_EnableAlarm := #I_EnHHHAlarm,
                  I_AlarmResetPB := #I_ResHHHAlarm,
                  O_Alarm => #HHHAlarm,
                  O_AlarmABCondition => #HHHAlarmAlmCond);
   END_IF;
END_REGION

REGION Network 3: **** 2.2 - Alarms - Alarm generation **** Alarm High High Limit
   // Alarm High High Limit
   IF "TRUE" THEN
       #HH_Alarm(I_Input := #HHTempSR,   // "LProc1AlarmMultiIn"
                 I_AlarmClass := 'A',
                 I_EnableAlarm := #I_EnHHAlarm,
                 I_AlarmResetPB := #I_ResHHAlarm,
                 O_Alarm => #HHAlarm,
                 O_AlarmABCondition => #HHAlarmAlmCond);
   END_IF;
END_REGION

REGION Network 4: **** 2.2 - Alarms - Alarm generation **** Alarm High Limit
   // Alarm High Limit
   IF "TRUE" THEN
       #H_Alarm(I_Input := #HTempSR,   // "LProc1AlarmMultiIn"
                I_AlarmClass := 'A',
                I_EnableAlarm := #I_EnHAlarm,
                I_AlarmResetPB := #I_ResHAlarm,
                O_Alarm => #HAlarm,
                O_AlarmABCondition => #HAlarmAlmCond);
   END_IF;
END_REGION

REGION Network 5: **** 2.2 - Alarms - Alarm generation **** Alarm Low Limit
   // Alarm Low Limit
   IF "TRUE" THEN
       #L_Alarm(I_Input := #LTempSR,   // "LProc1AlarmMultiIn"
                I_AlarmClass := 'A',
                I_EnableAlarm := #I_EnLAlarm,
                I_AlarmResetPB := #I_ResLAlarm,
                O_Alarm => #LAlarm,
                O_AlarmABCondition => #LAlarmAlmCond);
   END_IF;
END_REGION

REGION Network 6: **** 2.2 - Alarms - Alarm generation **** Alarm Low Low Limit
   // Alarm Low Low Limit
   IF "TRUE" THEN
       #LL_Alarm(I_Input := #LLTempSR,   // "LProc1AlarmMultiIn"
                 I_AlarmClass := 'A',
                 I_EnableAlarm := #I_EnLLAlarm,
                 I_AlarmResetPB := #I_ResLLAlarm,
                 O_Alarm => #LLAlarm,
                 O_AlarmABCondition => #LLAlarmAlmCond);
   END_IF;
END_REGION

REGION Network 7: **** 2.2 - Alarms - Alarm generation **** Alarm Low Low Low Limit
   // Alarm Low Low Low Limit
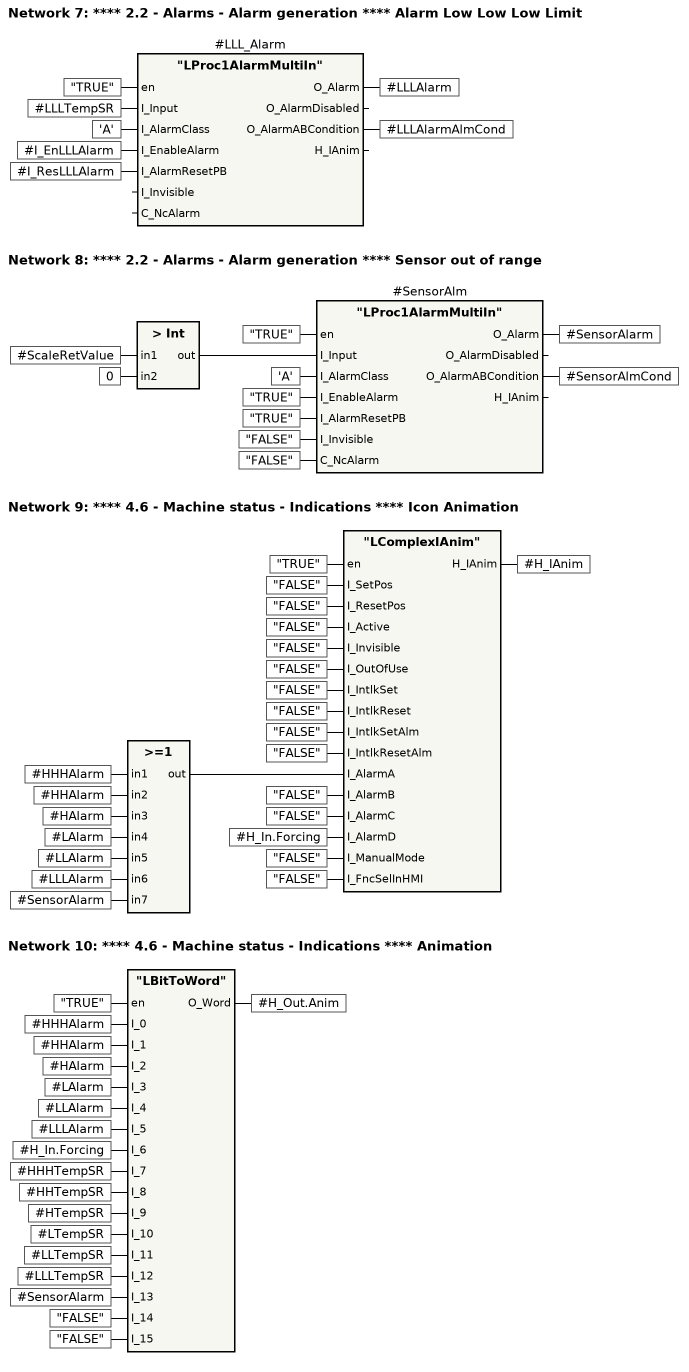
   IF "TRUE" THEN
       #LLL_Alarm(I_Input := #LLLTempSR,   // "LProc1AlarmMultiIn"
                  I_AlarmClass := 'A',
                  I_EnableAlarm := #I_EnLLLAlarm,
                  I_AlarmResetPB := #I_ResLLLAlarm,
                  O_Alarm => #LLLAlarm,
                  O_AlarmABCondition => #LLLAlarmAlmCond);
   END_IF;
END_REGION

REGION Network 8: **** 2.2 - Alarms - Alarm generation **** Sensor out of range
   // Sensor out of range
   IF "TRUE" THEN
       #SensorAlm(I_Input := #ScaleRetValue > 0,   // "LProc1AlarmMultiIn"
                  I_AlarmClass := 'A',
                  I_EnableAlarm := "TRUE",
                  I_AlarmResetPB := "TRUE",
                  I_Invisible := "FALSE",
                  C_NcAlarm := "FALSE",
                  O_Alarm => #SensorAlarm,
                  O_AlarmABCondition => #SensorAlmCond);
   END_IF;
END_REGION

REGION Network 9: **** 4.6 - Machine status - Indications **** Icon Animation
   // Icon Animation
   IF "TRUE" THEN
       "LComplexIAnim"(I_SetPos := "FALSE",
                       I_ResetPos := "FALSE",
                       I_Active := "FALSE",
                       I_Invisible := "FALSE",
                       I_OutOfUse := "FALSE",
                       I_IntlkSet := "FALSE",
                       I_IntlkReset := "FALSE",
                       I_IntlkSetAlm := "FALSE",
                       I_IntlkResetAlm := "FALSE",
                       I_AlarmA := #HHHAlarm OR #HHAlarm OR #HAlarm OR #LAlarm OR #LLAlarm OR #LLLAlarm OR #SensorAlarm,
                       I_AlarmB := "FALSE",
                       I_AlarmC := "FALSE",
                       I_AlarmD := #H_In.Forcing,
                       I_ManualMode := "FALSE",
                       I_FncSelInHMI := "FALSE",
                       H_IAnim => #H_IAnim);
   END_IF;
END_REGION

REGION Network 10: **** 4.6 - Machine status - Indications **** Animation
   // Animation
   IF "TRUE" THEN
       "LBitToWord"(I_0 := #HHHAlarm,
                    I_1 := #HHAlarm,
                    I_2 := #HAlarm,
                    I_3 := #LAlarm,
                    I_4 := #LLAlarm,
                    I_5 := #LLLAlarm,
                    I_6 := #H_In.Forcing,
                    I_7 := #HHHTempSR,
                    I_8 := #HHTempSR,
                    I_9 := #HTempSR,
                    I_10 := #LTempSR,
                    I_11 := #LLTempSR,
                    I_12 := #LLLTempSR,
                    I_13 := #SensorAlarm,
                    I_14 := "FALSE",
                    I_15 := "FALSE",
                    O_Word => #H_Out.Anim);
   END_IF;
END_REGION

REGION Network 11: **** 4.6 - Machine status - Indications **** Animation DB number
   // Animation DB number
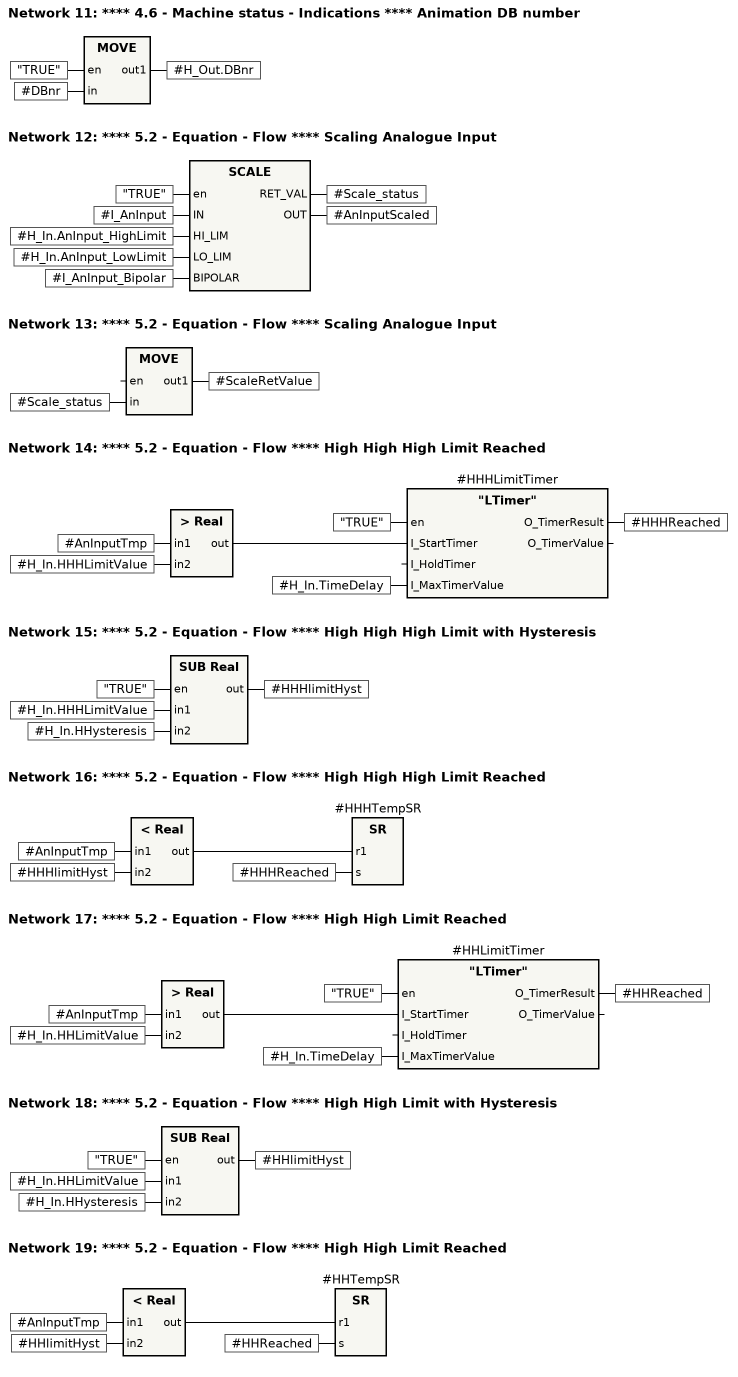
   IF "TRUE" THEN #H_Out.DBnr := #DBnr; END_IF;
END_REGION

REGION Network 12: **** 5.2 - Equation - Flow **** Scaling Analogue Input
   // Scaling Analogue Input
   IF "TRUE" THEN
       #Scale_status := SCALE(IN := #I_AnInput,
                              HI_LIM := #H_In.AnInput_HighLimit,
                              LO_LIM := #H_In.AnInput_LowLimit,
                              BIPOLAR := #I_AnInput_Bipolar,
                              OUT => #AnInputScaled);
   END_IF;
END_REGION

REGION Network 13: **** 5.2 - Equation - Flow **** Scaling Analogue Input
   // Scaling Analogue Input
   #ScaleRetValue := #Scale_status;
END_REGION

REGION Network 14: **** 5.2 - Equation - Flow **** High High High Limit Reached
   // High High High Limit Reached
   IF "TRUE" THEN
       #HHHLimitTimer(I_StartTimer := #AnInputTmp > #H_In.HHHLimitValue,   // "LTimer"
                      I_MaxTimerValue := #H_In.TimeDelay,
                      O_TimerResult => #HHHReached);
   END_IF;
END_REGION

REGION Network 15: **** 5.2 - Equation - Flow **** High High High Limit with Hysteresis
   // High High High Limit with Hysteresis
   IF "TRUE" THEN #HHHlimitHyst := #H_In.HHHLimitValue - #H_In.HHysteresis; END_IF;
END_REGION

REGION Network 16: **** 5.2 - Equation - Flow **** High High High Limit Reached
   // High High High Limit Reached
   IF #HHHReached THEN
       #HHHTempSR := TRUE;   // SR flip-flop
   END_IF;
   IF #AnInputTmp < #HHHlimitHyst THEN #HHHTempSR := FALSE; END_IF;
END_REGION

REGION Network 17: **** 5.2 - Equation - Flow **** High High Limit Reached
   // High High Limit Reached
   IF "TRUE" THEN
       #HHLimitTimer(I_StartTimer := #AnInputTmp > #H_In.HHLimitValue,   // "LTimer"
                     I_MaxTimerValue := #H_In.TimeDelay,
                     O_TimerResult => #HHReached);
   END_IF;
END_REGION

REGION Network 18: **** 5.2 - Equation - Flow **** High High Limit with Hysteresis
   // High High Limit with Hysteresis
   IF "TRUE" THEN #HHlimitHyst := #H_In.HHLimitValue - #H_In.HHysteresis; END_IF;
END_REGION

REGION Network 19: **** 5.2 - Equation - Flow **** High High Limit Reached
   // High High Limit Reached
   IF #HHReached THEN
       #HHTempSR := TRUE;   // SR flip-flop
   END_IF;
   IF #AnInputTmp < #HHlimitHyst THEN #HHTempSR := FALSE; END_IF;
END_REGION

REGION Network 20: **** 5.2 - Equation - Flow **** High Limit Reached
   // High Limit Reached
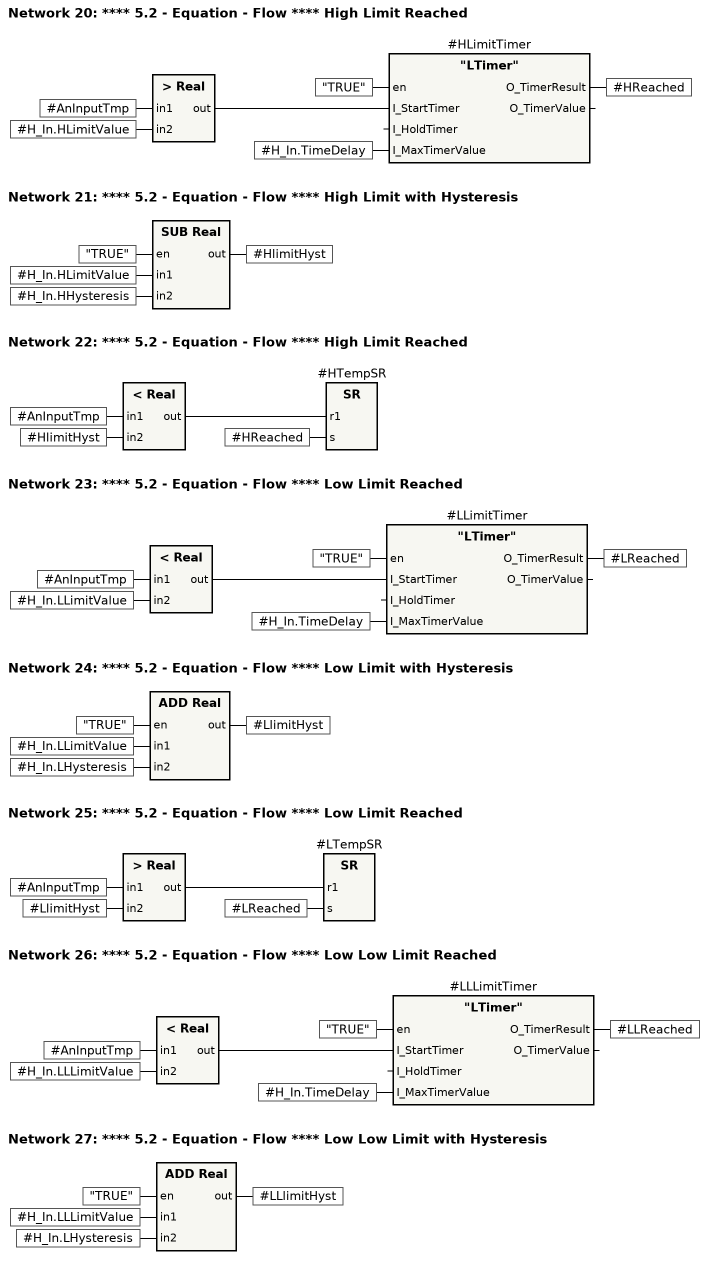
   IF "TRUE" THEN
       #HLimitTimer(I_StartTimer := #AnInputTmp > #H_In.HLimitValue,   // "LTimer"
                    I_MaxTimerValue := #H_In.TimeDelay,
                    O_TimerResult => #HReached);
   END_IF;
END_REGION

REGION Network 21: **** 5.2 - Equation - Flow **** High Limit with Hysteresis
   // High Limit with Hysteresis
   IF "TRUE" THEN #HlimitHyst := #H_In.HLimitValue - #H_In.HHysteresis; END_IF;
END_REGION

REGION Network 22: **** 5.2 - Equation - Flow **** High Limit Reached
   // High Limit Reached
   IF #HReached THEN
       #HTempSR := TRUE;   // SR flip-flop
   END_IF;
   IF #AnInputTmp < #HlimitHyst THEN #HTempSR := FALSE; END_IF;
END_REGION

REGION Network 23: **** 5.2 - Equation - Flow **** Low Limit Reached
   // Low Limit Reached
   IF "TRUE" THEN
       #LLimitTimer(I_StartTimer := #AnInputTmp < #H_In.LLimitValue,   // "LTimer"
                    I_MaxTimerValue := #H_In.TimeDelay,
                    O_TimerResult => #LReached);
   END_IF;
END_REGION

REGION Network 24: **** 5.2 - Equation - Flow **** Low Limit with Hysteresis
   // Low Limit with Hysteresis
   IF "TRUE" THEN #LlimitHyst := #H_In.LLimitValue + #H_In.LHysteresis; END_IF;
END_REGION

REGION Network 25: **** 5.2 - Equation - Flow **** Low Limit Reached
   // Low Limit Reached
   IF #LReached THEN
       #LTempSR := TRUE;   // SR flip-flop
   END_IF;
   IF #AnInputTmp > #LlimitHyst THEN #LTempSR := FALSE; END_IF;
END_REGION

REGION Network 26: **** 5.2 - Equation - Flow **** Low Low Limit Reached
   // Low Low Limit Reached
   IF "TRUE" THEN
       #LLLimitTimer(I_StartTimer := #AnInputTmp < #H_In.LLLimitValue,   // "LTimer"
                     I_MaxTimerValue := #H_In.TimeDelay,
                     O_TimerResult => #LLReached);
   END_IF;
END_REGION

REGION Network 27: **** 5.2 - Equation - Flow **** Low Low Limit with Hysteresis
   // Low Low Limit with Hysteresis
   IF "TRUE" THEN #LLlimitHyst := #H_In.LLLimitValue + #H_In.LHysteresis; END_IF;
END_REGION

REGION Network 28: **** 5.2 - Equation - Flow **** Low Low Limit Reached
   // Low Low Limit Reached
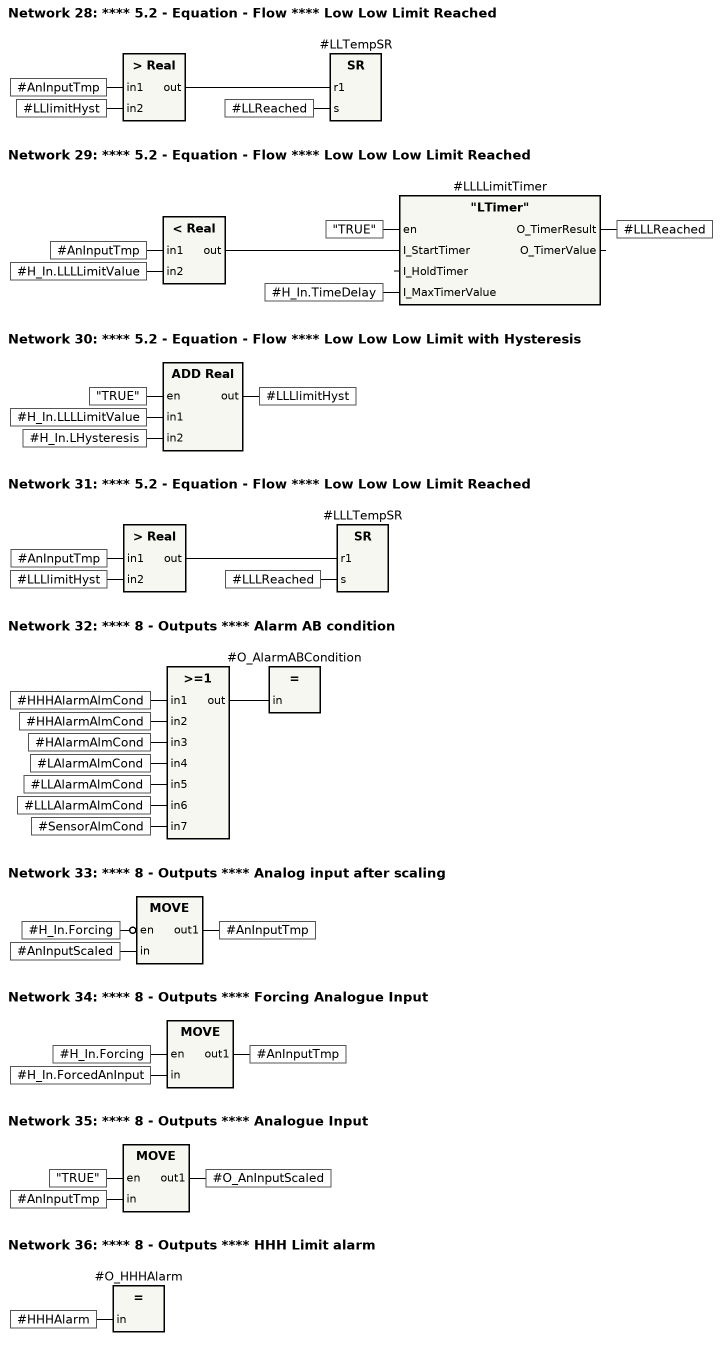
   IF #LLReached THEN
       #LLTempSR := TRUE;   // SR flip-flop
   END_IF;
   IF #AnInputTmp > #LLlimitHyst THEN #LLTempSR := FALSE; END_IF;
END_REGION

REGION Network 29: **** 5.2 - Equation - Flow **** Low Low Low Limit Reached
   // Low Low Low Limit Reached
   IF "TRUE" THEN
       #LLLLimitTimer(I_StartTimer := #AnInputTmp < #H_In.LLLLimitValue,   // "LTimer"
                      I_MaxTimerValue := #H_In.TimeDelay,
                      O_TimerResult => #LLLReached);
   END_IF;
END_REGION

REGION Network 30: **** 5.2 - Equation - Flow **** Low Low Low Limit with Hysteresis
   // Low Low Low Limit with Hysteresis
   IF "TRUE" THEN #LLLlimitHyst := #H_In.LLLLimitValue + #H_In.LHysteresis; END_IF;
END_REGION

REGION Network 31: **** 5.2 - Equation - Flow **** Low Low Low Limit Reached
   // Low Low Low Limit Reached
   IF #LLLReached THEN
       #LLLTempSR := TRUE;   // SR flip-flop
   END_IF;
   IF #AnInputTmp > #LLLlimitHyst THEN #LLLTempSR := FALSE; END_IF;
END_REGION

REGION Network 32: **** 8 - Outputs **** Alarm AB condition
   // Alarm AB condition
   #O_AlarmABCondition := #HHHAlarmAlmCond OR #HHAlarmAlmCond OR #HAlarmAlmCond OR #LAlarmAlmCond OR #LLAlarmAlmCond OR #LLLAlarmAlmCond OR #SensorAlmCond;
END_REGION

REGION Network 33: **** 8 - Outputs **** Analog input after scaling
   // Analog input after scaling
   IF NOT #H_In.Forcing THEN #AnInputTmp := #AnInputScaled; END_IF;
END_REGION

REGION Network 34: **** 8 - Outputs **** Forcing Analogue Input
   // Forcing Analogue Input
   IF #H_In.Forcing THEN #AnInputTmp := #H_In.ForcedAnInput; END_IF;
END_REGION

REGION Network 35: **** 8 - Outputs **** Analogue Input
   // Analogue Input
   IF "TRUE" THEN #O_AnInputScaled := #AnInputTmp; END_IF;
END_REGION

REGION Network 36: **** 8 - Outputs **** HHH Limit alarm
   // HHH Limit alarm
   #O_HHHAlarm := #HHHAlarm;
END_REGION

REGION Network 37: **** 8 - Outputs **** HH Limit alarm
   // HH Limit alarm
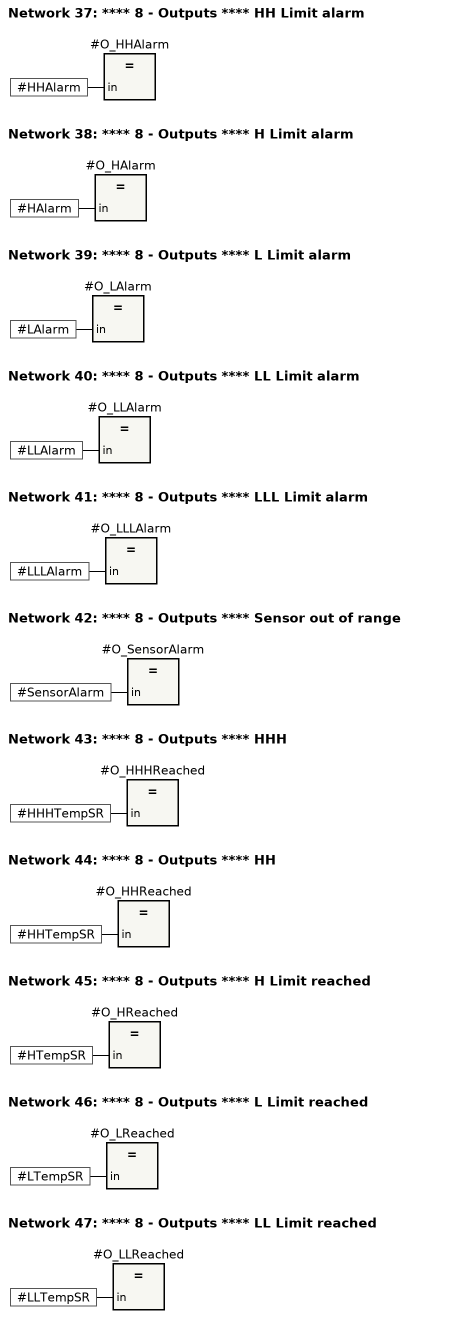
   #O_HHAlarm := #HHAlarm;
END_REGION

REGION Network 38: **** 8 - Outputs **** H Limit alarm
   // H Limit alarm
   #O_HAlarm := #HAlarm;
END_REGION

REGION Network 39: **** 8 - Outputs **** L Limit alarm
   // L Limit alarm
   #O_LAlarm := #LAlarm;
END_REGION

REGION Network 40: **** 8 - Outputs **** LL Limit alarm
   // LL Limit alarm
   #O_LLAlarm := #LLAlarm;
END_REGION

REGION Network 41: **** 8 - Outputs **** LLL Limit alarm
   // LLL Limit alarm
   #O_LLLAlarm := #LLLAlarm;
END_REGION

REGION Network 42: **** 8 - Outputs **** Sensor out of range
   // Sensor out of range
   #O_SensorAlarm := #SensorAlarm;
END_REGION

REGION Network 43: **** 8 - Outputs **** HHH
   // HHH
   //  Limit reached
   #O_HHHReached := #HHHTempSR;
END_REGION

REGION Network 44: **** 8 - Outputs **** HH
   // HH
   //  Limit reached
   #O_HHReached := #HHTempSR;
END_REGION

REGION Network 45: **** 8 - Outputs **** H Limit reached
   // H Limit reached
   #O_HReached := #HTempSR;
END_REGION

REGION Network 46: **** 8 - Outputs **** L Limit reached
   // L Limit reached
   #O_LReached := #LTempSR;
END_REGION

REGION Network 47: **** 8 - Outputs **** LL Limit reached
   // LL Limit reached
   #O_LLReached := #LLTempSR;
END_REGION

REGION Network 48: **** 8 - Outputs **** LLL Limit reached
   // LLL Limit reached
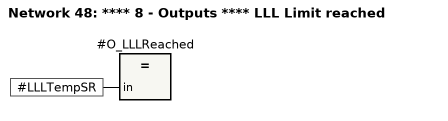
   #O_LLLReached := #LLLTempSR;
END_REGION
END_FUNCTION_BLOCK

FUNCTION_BLOCK "LProc1AlarmMultiIn"   // FB1737, FBD
TITLE = L1AlarmMultiIn / LProc1AlarmMultiIn
{ S7_Optimized_Access := 'FALSE' }
AUTHOR : VCC
FAMILY : AlarmHnd
NAME : 1Alarm
VERSION : 1.0
// ================================================================================
// This module is used inside another FB where one alarm shall be generated when 
// one (security) input becomes True.
// The alarm can be True only when the input Enable Alarm is also True.
// The alarm can be True only when the input Disable Alarm is False. When the 
// alarm is disabled from HMI, a boolean output is available to inform the upper 
// level and do action in the Alarm summary.
// When the conditions to generate the alarm disappear, a boolean output is 
// available to inform the upper level that the alarm can be reset.
// The alarm is reset by means of the AlarmResetPB signal.
// ================================================================================
// stored: AutoNumber false, IsIECCheckEnabled false, SetENOAutomatically False, UDAEnableTagReadback false
   VAR_INPUT
      I_Input { ExternalAccessible := 'False'; ExternalVisible := 'False'; ExternalWritable := 'False'} : Bool;   // Input signal of the alarm
      I_AlarmClass { ExternalAccessible := 'False'; ExternalVisible := 'False'; ExternalWritable := 'False'} : Char;   // Alarm class -> A - B - C - D or E
      I_EnableAlarm { ExternalAccessible := 'False'; ExternalVisible := 'False'; ExternalWritable := 'False'} : Bool := TRUE;   // Enable alarm from upper level
      I_AlarmResetPB { ExternalAccessible := 'False'; ExternalVisible := 'False'; ExternalWritable := 'False'} : Bool;   // Alarm reset pushbutton is activated
      I_Invisible { ExternalAccessible := 'False'; ExternalVisible := 'False'; ExternalWritable := 'False'} : Bool;   // Invisible
      C_NcAlarm { ExternalAccessible := 'False'; ExternalVisible := 'False'; ExternalWritable := 'False'} : Bool;   // Alarm contact NC
   END_VAR
   VAR_OUTPUT
      O_Alarm { ExternalAccessible := 'False'; ExternalVisible := 'False'; ExternalWritable := 'False'} : Bool;   // Alarm
      O_AlarmDisabled { ExternalAccessible := 'False'; ExternalVisible := 'False'; ExternalWritable := 'False'} : Bool;   // Alarm disabled from HMI
      O_AlarmABCondition { ExternalAccessible := 'False'; ExternalVisible := 'False'; ExternalWritable := 'False'} : Bool;   // Alarm AB condition
      H_IAnim { ExternalAccessible := 'False'; ExternalVisible := 'False'; ExternalWritable := 'False'} : Word;
   END_VAR
   VAR DB_SPECIFIC
      H_In : Struct   // HMI
         DisableAlarm : Bool;   // Disable alarm from HMI
      END_STRUCT;
      H_Out : Struct   // HMI
         DBnr : Int;   // HMI Animation DB number
      END_STRUCT;
      Alarm { ExternalAccessible := 'False'; ExternalVisible := 'False'; ExternalWritable := 'False'} : Bool;   // Alarm
      AlarmClass_A { ExternalAccessible := 'False'; ExternalVisible := 'False'; ExternalWritable := 'False'} : Bool;   // The alarm is from alarm class A
      AlarmClass_B { ExternalAccessible := 'False'; ExternalVisible := 'False'; ExternalWritable := 'False'} : Bool;   // The alarm is from alarm class B
      AlarmClass_C { ExternalAccessible := 'False'; ExternalVisible := 'False'; ExternalWritable := 'False'} : Bool;   // The alarm is from alarm class C
      AlarmClass_D { ExternalAccessible := 'False'; ExternalVisible := 'False'; ExternalWritable := 'False'} : Bool;   // The alarm is from alarm class D
      AlarmClass_E { ExternalAccessible := 'False'; ExternalVisible := 'False'; ExternalWritable := 'False'} : Bool;   // The alarm is from alarm class E
      AlarmCond { ExternalAccessible := 'False'; ExternalVisible := 'False'; ExternalWritable := 'False'} : Bool;   // Alarm condition
      DBnr { ExternalAccessible := 'False'; ExternalVisible := 'False'; ExternalWritable := 'False'} : Int;   // HMI DB number
   END_VAR
BEGIN

NETWORK
TITLE = **** 1 - Inputs **** DB number
// DB number
      L     DINO;
      T     #DBnr;

NETWORK
TITLE = **** 1 - Inputs **** Alarm class
// Alarm class
// Alarm class = E
      L     #I_AlarmClass;
      L     'E';
      ==I;
      =     #AlarmClass_E;

// Alarm class = D
      L     #I_AlarmClass;
      L     'D';
      ==I;
      =     #AlarmClass_D;

// Alarm class = C
      L     #I_AlarmClass;
      L     'C';
      ==I;
      =     #AlarmClass_C;

// Alarm class = B
      L     #I_AlarmClass;
      L     'B';
      ==I;
      =     #AlarmClass_B;

// Alarm class = A
      AN    #AlarmClass_B;
      AN    #AlarmClass_C;
      AN    #AlarmClass_D;
      AN    #AlarmClass_E;
      =     #AlarmClass_A;


REGION Network 3: **** 2.2 - Alarms - Alarms Generation **** Alarm Condition
   // Condition for the Alarm
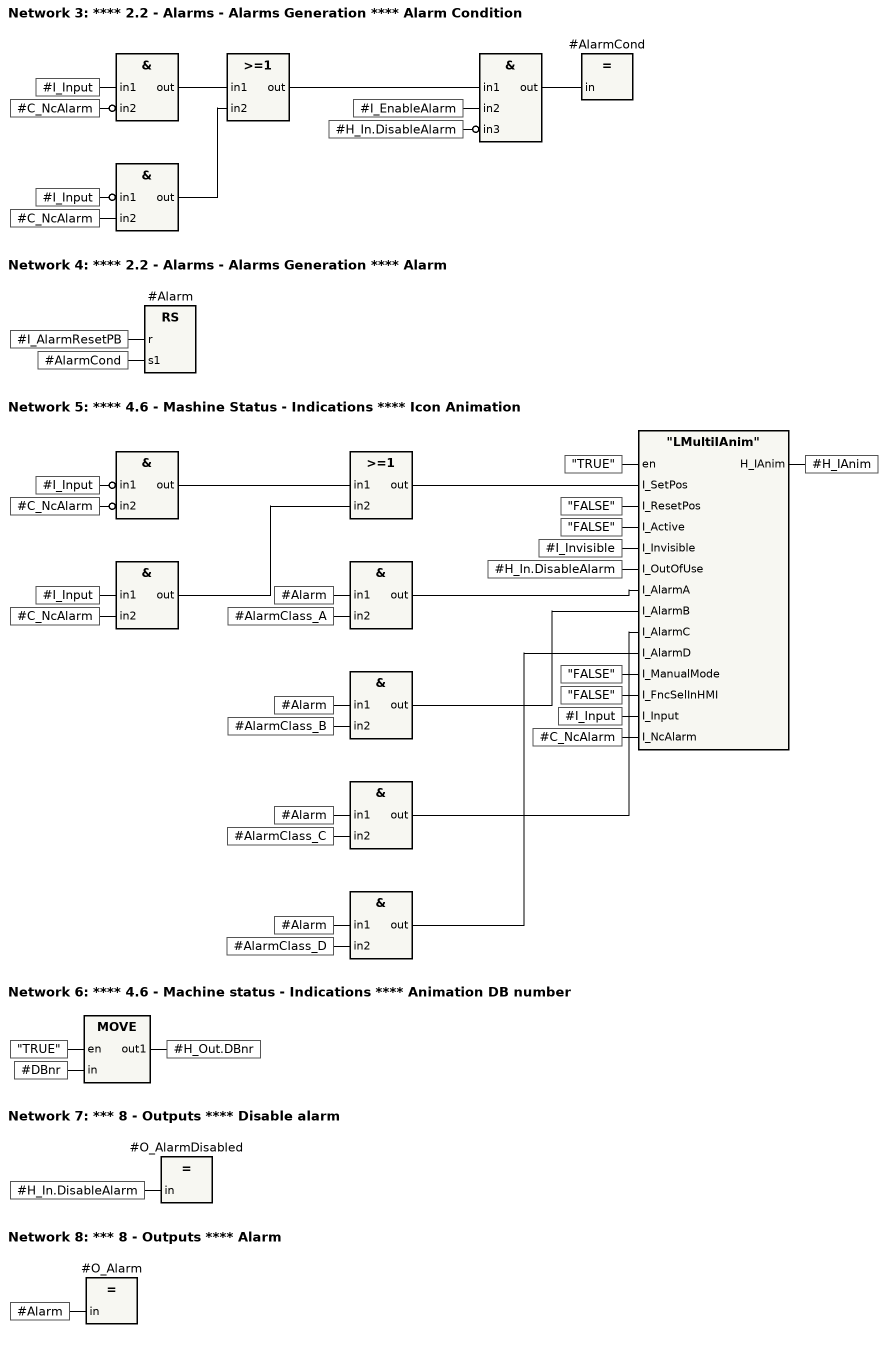
   #AlarmCond := ((#I_Input AND NOT #C_NcAlarm) OR (NOT #I_Input AND #C_NcAlarm)) AND #I_EnableAlarm AND NOT #H_In.DisableAlarm;
END_REGION

REGION Network 4: **** 2.2 - Alarms - Alarms Generation **** Alarm
   // Creation of the Alarm
   IF #I_AlarmResetPB THEN
       #Alarm := FALSE;   // RS flip-flop
   END_IF;
   IF #AlarmCond THEN #Alarm := TRUE; END_IF;
END_REGION

REGION Network 5: **** 4.6 - Mashine Status - Indications **** Icon Animation
   // Icon Animation
   IF "TRUE" THEN
       "LMultiIAnim"(I_SetPos := (NOT #I_Input AND NOT #C_NcAlarm) OR (#I_Input AND #C_NcAlarm),
                     I_ResetPos := "FALSE",
                     I_Active := "FALSE",
                     I_Invisible := #I_Invisible,
                     I_OutOfUse := #H_In.DisableAlarm,
                     I_AlarmA := #Alarm AND #AlarmClass_A,
                     I_AlarmB := #Alarm AND #AlarmClass_B,
                     I_AlarmC := #Alarm AND #AlarmClass_C,
                     I_AlarmD := #Alarm AND #AlarmClass_D,
                     I_ManualMode := "FALSE",
                     I_FncSelInHMI := "FALSE",
                     I_Input := #I_Input,
                     I_NcAlarm := #C_NcAlarm,
                     H_IAnim => #H_IAnim);
   END_IF;
END_REGION

REGION Network 6: **** 4.6 - Machine status - Indications **** Animation DB number
   IF "TRUE" THEN #H_Out.DBnr := #DBnr; END_IF;
END_REGION

REGION Network 7: *** 8 - Outputs **** Disable alarm
   // Alarm disabled from HMI
   #O_AlarmDisabled := #H_In.DisableAlarm;
END_REGION

REGION Network 8: *** 8 - Outputs **** Alarm
   // Output of the Alarm
   #O_Alarm := #Alarm;
END_REGION

REGION Network 9: **** 8 - Outputs **** Alarm AB Condition
   // Alarm Resetable
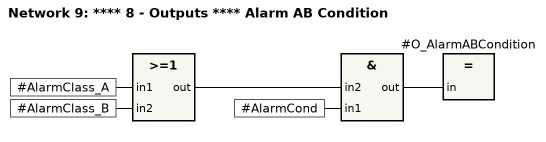
   #O_AlarmABCondition := (#AlarmClass_A OR #AlarmClass_B) AND #AlarmCond;
END_REGION
END_FUNCTION_BLOCK

FUNCTION_BLOCK "LProcMonStabValv"   // FB1701, FBD
TITLE = LProcMonStabValv
{ S7_Optimized_Access := 'FALSE' }
AUTHOR : VCC
FAMILY : ProcEqp
NAME : ProcValv
VERSION : 1.0
// ================================================================================
// This module is used to activate a monostable valve. It includes its own Mode 
// function. There is the possibility to use it normally open or normally closed, 
// with or without closed and open detections.
// ================================================================================
// stored: AutoNumber false, IsIECCheckEnabled false, SetENOAutomatically False, UDAEnableTagReadback false
   VAR_INPUT
      I_MaxTime { ExternalAccessible := 'False'; ExternalVisible := 'False'; ExternalWritable := 'False'} : DInt;   // Maximum Time to get Set and reset detections
      I_DetSet { ExternalAccessible := 'False'; ExternalVisible := 'False'; ExternalWritable := 'False'} : Bool;   // Detection SET
      I_DetReset { ExternalAccessible := 'False'; ExternalVisible := 'False'; ExternalWritable := 'False'} : Bool;   // Detection RESET
      I_EnableAlarm { ExternalAccessible := 'False'; ExternalVisible := 'False'; ExternalWritable := 'False'} : Bool;   // Enable Alarm for the Acof detections
      I_AutoReq { ExternalAccessible := 'False'; ExternalVisible := 'False'; ExternalWritable := 'False'} : Bool;   // Auto Request from equation or Sequence
      I_InterlockOk { ExternalAccessible := 'False'; ExternalVisible := 'False'; ExternalWritable := 'False'} : Bool;   // Interlock
      I_PBSetPBResetAllAutoSel { ExternalAccessible := 'False'; ExternalVisible := 'False'; ExternalWritable := 'False'} : Struct   // Set PB activated - Reset PB activated - All HMI Auto selected
         HMI1SetPB { ExternalAccessible := 'False'; ExternalVisible := 'False'; ExternalWritable := 'False'} : Bool;   // Set PB activated on HMI1
         HMI1ResetPB { ExternalAccessible := 'False'; ExternalVisible := 'False'; ExternalWritable := 'False'} : Bool;   // Reset PB activated on HMI1
         HMI1AllHMIAutoSel { ExternalAccessible := 'False'; ExternalVisible := 'False'; ExternalWritable := 'False'} : Bool;   // All HMI Auto selected on HMI1
         HMI2SetPB { ExternalAccessible := 'False'; ExternalVisible := 'False'; ExternalWritable := 'False'} : Bool;   // Set PB activated on HMI2
         HMI2ResetPB { ExternalAccessible := 'False'; ExternalVisible := 'False'; ExternalWritable := 'False'} : Bool;   // Reset PB activated on HMI2
         HMI2AllHMIAutoSel { ExternalAccessible := 'False'; ExternalVisible := 'False'; ExternalWritable := 'False'} : Bool;   // All HMI Auto selected on HMI2
         HMI3SetPB { ExternalAccessible := 'False'; ExternalVisible := 'False'; ExternalWritable := 'False'} : Bool;   // Set PB activated on HMI3
         HMI3ResetPB { ExternalAccessible := 'False'; ExternalVisible := 'False'; ExternalWritable := 'False'} : Bool;   // Reset PB activated on HMI3
         HMI3AllHMIAutoSel { ExternalAccessible := 'False'; ExternalVisible := 'False'; ExternalWritable := 'False'} : Bool;   // All HMI Auto selected on HMI3
         HMI4SetPB { ExternalAccessible := 'False'; ExternalVisible := 'False'; ExternalWritable := 'False'} : Bool;   // Set PB activated on HMI4
         HMI4ResetPB { ExternalAccessible := 'False'; ExternalVisible := 'False'; ExternalWritable := 'False'} : Bool;   // Reset PB activated on HMI4
         HMI4AllHMIAutoSel { ExternalAccessible := 'False'; ExternalVisible := 'False'; ExternalWritable := 'False'} : Bool;   // All HMI Auto selected on HMI4
         HMI5SetPB { ExternalAccessible := 'False'; ExternalVisible := 'False'; ExternalWritable := 'False'} : Bool;   // Set PB activated on HMI5
         HMI5ResetPB { ExternalAccessible := 'False'; ExternalVisible := 'False'; ExternalWritable := 'False'} : Bool;   // Reset PB activated on HMI5
         HMI5AllHMIAutoSel { ExternalAccessible := 'False'; ExternalVisible := 'False'; ExternalWritable := 'False'} : Bool;   // All HMI Auto selected on HMI5
         StartPBSel { ExternalAccessible := 'False'; ExternalVisible := 'False'; ExternalWritable := 'False'} : Bool;   // Start is activated
         AlarmResetPBSel { ExternalAccessible := 'False'; ExternalVisible := 'False'; ExternalWritable := 'False'} : Bool;   // Alarm reset is activated
      END_STRUCT;
      I_UpperLevelAlarmA { ExternalAccessible := 'False'; ExternalVisible := 'False'; ExternalWritable := 'False'} : Bool;   // Alarm A active from the top level
      I_UpperLevelAlarmB { ExternalAccessible := 'False'; ExternalVisible := 'False'; ExternalWritable := 'False'} : Bool;   // Alarm B active from the top level
      C_EnableSetResetHMI { ExternalAccessible := 'False'; ExternalVisible := 'False'; ExternalWritable := 'False'} : Bool;   // Enable Set-Reset functions from HMI
      C_ManualForcedUsed { ExternalAccessible := 'False'; ExternalVisible := 'False'; ExternalWritable := 'False'} : Bool;   // Manual Forced is used (=true)
      C_SelfHolding { ExternalAccessible := 'False'; ExternalVisible := 'False'; ExternalWritable := 'False'} : Bool := TRUE;   // Enable SelfHolding Command
      C_DetSetUsed { ExternalAccessible := 'False'; ExternalVisible := 'False'; ExternalWritable := 'False'} : Bool;   // Detection SET used (true=used)
      C_DetResetUsed { ExternalAccessible := 'False'; ExternalVisible := 'False'; ExternalWritable := 'False'} : Bool;   // Detection RESET used (true=used)
      C_ValveNO { ExternalAccessible := 'False'; ExternalVisible := 'False'; ExternalWritable := 'False'} : Bool;   // Valve Normally Open (NO=true)
   END_VAR
   VAR_OUTPUT
      O_ValveCmd { ExternalAccessible := 'False'; ExternalVisible := 'False'; ExternalWritable := 'False'} : Bool;   // Valve Command
      O_AlarmABCondition { ExternalAccessible := 'False'; ExternalVisible := 'False'; ExternalWritable := 'False'} : Bool;   // Alarm AB condition
      O_AlarmA { ExternalAccessible := 'False'; ExternalVisible := 'False'; ExternalWritable := 'False'} : Bool;   // Summary Alarm A from the Valve
      O_AlarmB { ExternalAccessible := 'False'; ExternalVisible := 'False'; ExternalWritable := 'False'} : Bool;   // Summary Alarm B from the Valve
      O_AlarmC { ExternalAccessible := 'False'; ExternalVisible := 'False'; ExternalWritable := 'False'} : Bool;   // Summary Alarm C from the Valve
      O_AlarmD { ExternalAccessible := 'False'; ExternalVisible := 'False'; ExternalWritable := 'False'} : Bool;   // Summary Alarm D from the Valve
      H_IAnim { ExternalAccessible := 'False'; ExternalVisible := 'False'; ExternalWritable := 'False'} : Word;   // HMI Animation of the icon
      H_AlarmWord { ExternalAccessible := 'False'; ExternalVisible := 'False'; ExternalWritable := 'False'} : DWord;   // Alarm Word
   END_VAR
   VAR DB_SPECIFIC
      AB_OverTimeAutoSel { ExternalAccessible := 'False'; ExternalVisible := 'False'; ExternalWritable := 'False'} : Bool;   // Alarm Overtime Auto selected
      AB_AcofDetSet { ExternalAccessible := 'False'; ExternalVisible := 'False'; ExternalWritable := 'False'} : Bool;   // Acof Fault Set detection
      AB_AcofDetReset { ExternalAccessible := 'False'; ExternalVisible := 'False'; ExternalWritable := 'False'} : Bool;   // Acof Fault Reset detection
      AD_InterlockAlarm { ExternalAccessible := 'False'; ExternalVisible := 'False'; ExternalWritable := 'False'} : Bool;   // Interlock Fault
      H_HMIModeCmd : Word;   // Mode commands from HMI
      H_ActiveHMI : Int;   // Active HMI
      H_NameActiveHMI : String[25];   // Name of the Active HMI
      H_Out : Struct   // HMI
         DetSetIAnim : Word;   // HMI Animation of the Detection
         DetResetIAnim : Word;   // HMI Animation of the Detection
         OutputIAnim : Word;   // HMI Animation of the output
         Anim : Word;   // HMI Animation of the object
         Anim2 : Word;   // HMI Animation of the object
         Anim3 : Bool;   // HMI Animation bool
         DBnr : Int;   // HMI Animation DB number
      END_STRUCT;
      OverTimeAutoSelCond { ExternalAccessible := 'False'; ExternalVisible := 'False'; ExternalWritable := 'False'} : Bool;   // Overtime Auto selected condition
      AcofDetSetCond { ExternalAccessible := 'False'; ExternalVisible := 'False'; ExternalWritable := 'False'} : Bool;   // Acof Detection set condition
      AcofDetResetCond { ExternalAccessible := 'False'; ExternalVisible := 'False'; ExternalWritable := 'False'} : Bool;   // Acof Detection reset condition
      AutoMode { ExternalAccessible := 'False'; ExternalVisible := 'False'; ExternalWritable := 'False'} : Bool;   // Auto mode
      ManualMode { ExternalAccessible := 'False'; ExternalVisible := 'False'; ExternalWritable := 'False'} : Bool;   // Manual mode
      AutoModeSel { ExternalAccessible := 'False'; ExternalVisible := 'False'; ExternalWritable := 'False'} : Bool;   // Auto Mode Selection from HMI
      ManualModeSel { ExternalAccessible := 'False'; ExternalVisible := 'False'; ExternalWritable := 'False'} : Bool;   // Manual Mode Selection from HMI
      ForcedMan { ExternalAccessible := 'False'; ExternalVisible := 'False'; ExternalWritable := 'False'} : Bool;   // Forced manual active
      ForcedManTimer { ExternalAccessible := 'False'; ExternalVisible := 'False'; ExternalWritable := 'False'} : Bool;   // Forced manual timer
      HMISetCmd { ExternalAccessible := 'False'; ExternalVisible := 'False'; ExternalWritable := 'False'} : Bool;   // Set Command on HMI
      HMIResetCmd { ExternalAccessible := 'False'; ExternalVisible := 'False'; ExternalWritable := 'False'} : Bool;   // Reset Command on HMI
      H_FncSelInHMI { ExternalAccessible := 'False'; ExternalVisible := 'False'; ExternalWritable := 'False'} : Bool;   // Manual selection from HMI
      SetPBMan { ExternalAccessible := 'False'; ExternalVisible := 'False'; ExternalWritable := 'False'} : Bool;   // Set pushbutton is activated in manual
      ResetPBMan { ExternalAccessible := 'False'; ExternalVisible := 'False'; ExternalWritable := 'False'} : Bool;   // Reset pushbutton is activated in manual
      AllHMIAutoSel { ExternalAccessible := 'False'; ExternalVisible := 'False'; ExternalWritable := 'False'} : Bool;   // All HMI Auto selected
      CmdRequest { ExternalAccessible := 'False'; ExternalVisible := 'False'; ExternalWritable := 'False'} : Bool;   // Command request to activate the component
      OvTimeAutoSel { ExternalAccessible := 'False'; ExternalVisible := 'False'; ExternalWritable := 'False'} : Bool;   // Alarm Overtime Auto selected and Component activated
      AlarmA { ExternalAccessible := 'False'; ExternalVisible := 'False'; ExternalWritable := 'False'} : Bool;   // Summation Alarm A of roller.
      AlarmB { ExternalAccessible := 'False'; ExternalVisible := 'False'; ExternalWritable := 'False'} : Bool;   // Summation Alarm B of roller.
      AlarmC { ExternalAccessible := 'False'; ExternalVisible := 'False'; ExternalWritable := 'False'} : Bool;   // Summation Alarm C of roller.
      AlarmD { ExternalAccessible := 'False'; ExternalVisible := 'False'; ExternalWritable := 'False'} : Bool;   // Summation Alarm D of roller.
      DBnr { ExternalAccessible := 'False'; ExternalVisible := 'False'; ExternalWritable := 'False'} : Int;   // HMI DB number
   END_VAR
   VAR
      DetSet { ExternalAccessible := 'False'; ExternalVisible := 'False'; ExternalWritable := 'False'; S7_SetPoint := 'True'} : "LProcAcofDet";   // Acof Detection Set
      DetReset { ExternalAccessible := 'False'; ExternalVisible := 'False'; ExternalWritable := 'False'; S7_SetPoint := 'True'} : "LProcAcofDet";   // Acof Detection Reset
      Modes { ExternalAccessible := 'False'; ExternalVisible := 'False'; ExternalWritable := 'False'; S7_SetPoint := 'True'} : "LProcObjectMode";
   END_VAR
   VAR DB_SPECIFIC
      CheckActiveHMI { ExternalAccessible := 'False'; ExternalVisible := 'False'; ExternalWritable := 'False'; S7_SetPoint := 'True'} : TP_TIME;   // Timer
      CheckActiveHMI_1 { ExternalAccessible := 'False'; ExternalVisible := 'False'; ExternalWritable := 'False'; S7_SetPoint := 'True'} : TP_TIME;   // Timer
      CheckActiveHMI_2 { ExternalAccessible := 'False'; ExternalVisible := 'False'; ExternalWritable := 'False'; S7_SetPoint := 'True'} : TON_TIME;   // Timer
      CheckActiveHMI_3 { ExternalAccessible := 'False'; ExternalVisible := 'False'; ExternalWritable := 'False'; S7_SetPoint := 'True'} : TON_TIME;   // Timer
   END_VAR
BEGIN

NETWORK
TITLE = **** 1 - Inputs **** DB number
// DB number
      L     DINO;
      T     #DBnr;

REGION Network 2: **** 2.2 - Alarms - Alarm Generation **** Interlock Alarm
   // Interlock Alarm
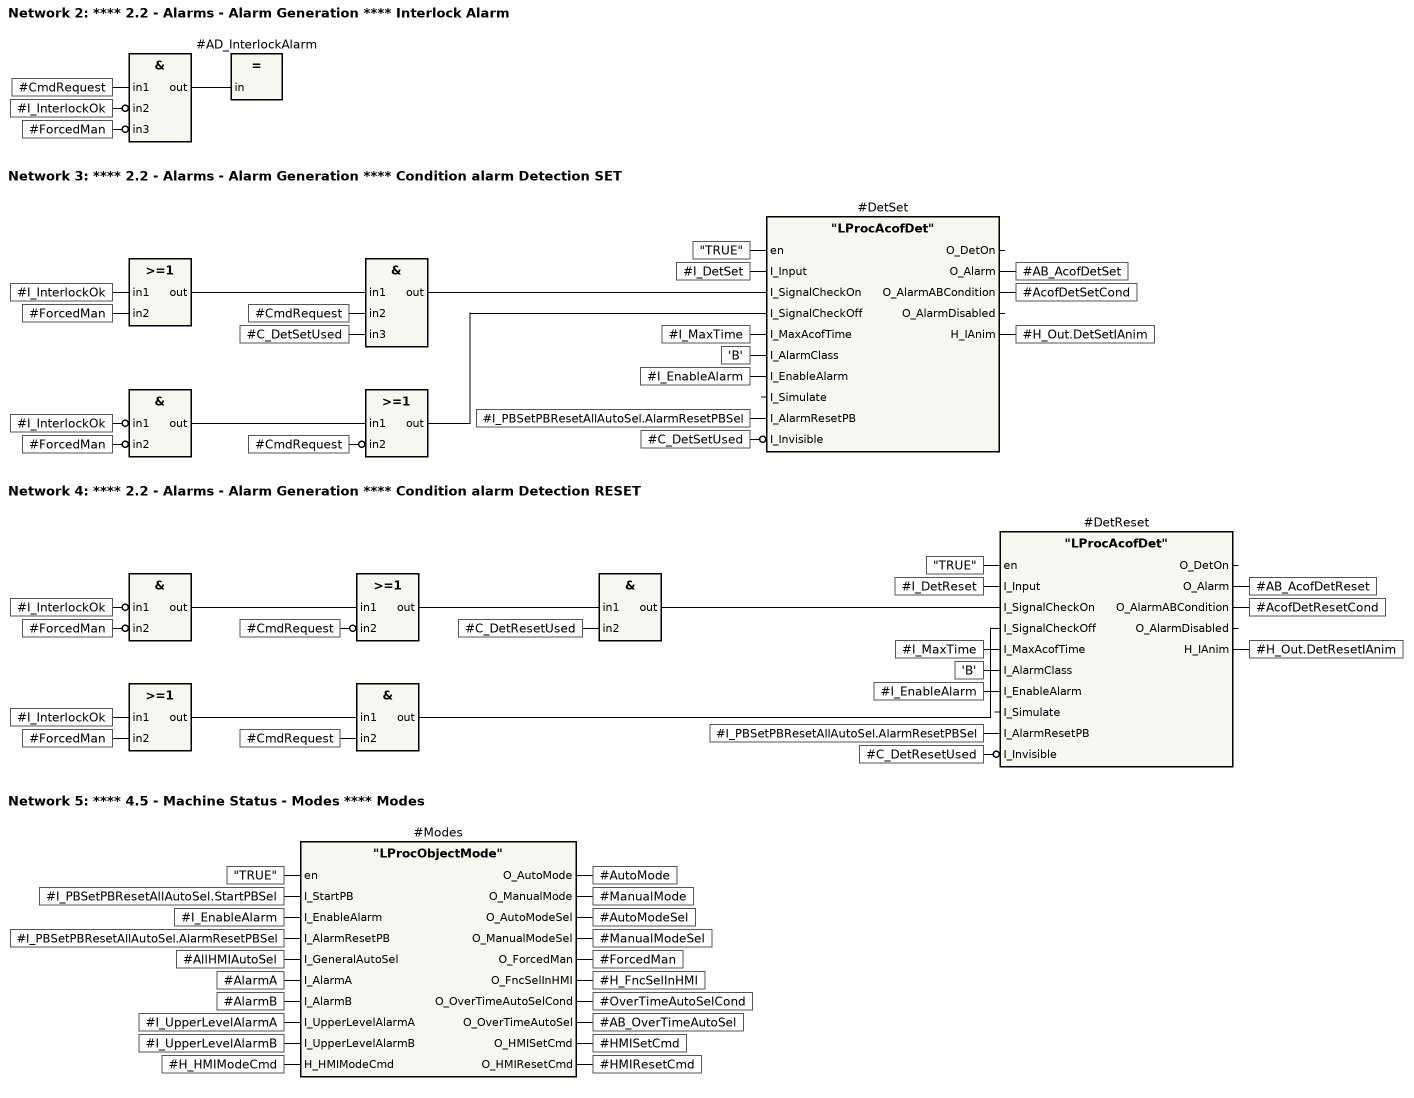
   #AD_InterlockAlarm := #CmdRequest AND NOT #I_InterlockOk AND NOT #ForcedMan;
END_REGION

REGION Network 3: **** 2.2 - Alarms - Alarm Generation **** Condition alarm Detection SET
   // Condition alarm Detection SET
   IF "TRUE" THEN
       #DetSet(I_Input := #I_DetSet,   // "LProcAcofDet"
               I_SignalCheckOn := (#I_InterlockOk OR #ForcedMan) AND #CmdRequest AND #C_DetSetUsed,
               I_SignalCheckOff := (NOT #I_InterlockOk AND NOT #ForcedMan) OR NOT #CmdRequest,
               I_MaxAcofTime := #I_MaxTime,
               I_AlarmClass := 'B',
               I_EnableAlarm := #I_EnableAlarm,
               I_AlarmResetPB := #I_PBSetPBResetAllAutoSel.AlarmResetPBSel,
               I_Invisible := NOT #C_DetSetUsed,
               O_Alarm => #AB_AcofDetSet,
               O_AlarmABCondition => #AcofDetSetCond,
               H_IAnim => #H_Out.DetSetIAnim);
   END_IF;
END_REGION

REGION Network 4: **** 2.2 - Alarms - Alarm Generation **** Condition alarm Detection RESET
   // Condition alarm Detection RESET
   IF "TRUE" THEN
       #DetReset(I_Input := #I_DetReset,   // "LProcAcofDet"
                 I_SignalCheckOn := ((NOT #I_InterlockOk AND NOT #ForcedMan) OR NOT #CmdRequest) AND #C_DetResetUsed,
                 I_SignalCheckOff := (#I_InterlockOk OR #ForcedMan) AND #CmdRequest,
                 I_MaxAcofTime := #I_MaxTime,
                 I_AlarmClass := 'B',
                 I_EnableAlarm := #I_EnableAlarm,
                 I_AlarmResetPB := #I_PBSetPBResetAllAutoSel.AlarmResetPBSel,
                 I_Invisible := NOT #C_DetResetUsed,
                 O_Alarm => #AB_AcofDetReset,
                 O_AlarmABCondition => #AcofDetResetCond,
                 H_IAnim => #H_Out.DetResetIAnim);
   END_IF;
END_REGION

REGION Network 5: **** 4.5 - Machine Status - Modes **** Modes
   // Modes
   IF "TRUE" THEN
       #Modes(I_StartPB := #I_PBSetPBResetAllAutoSel.StartPBSel,   // "LProcObjectMode"
              I_EnableAlarm := #I_EnableAlarm,
              I_AlarmResetPB := #I_PBSetPBResetAllAutoSel.AlarmResetPBSel,
              I_GeneralAutoSel := #AllHMIAutoSel,
              I_AlarmA := #AlarmA,
              I_AlarmB := #AlarmB,
              I_UpperLevelAlarmA := #I_UpperLevelAlarmA,
              I_UpperLevelAlarmB := #I_UpperLevelAlarmB,
              H_HMIModeCmd := #H_HMIModeCmd,
              O_AutoMode => #AutoMode,
              O_ManualMode => #ManualMode,
              O_AutoModeSel => #AutoModeSel,
              O_ManualModeSel => #ManualModeSel,
              O_ForcedMan => #ForcedMan,
              O_FncSelInHMI => #H_FncSelInHMI,
              O_OverTimeAutoSelCond => #OverTimeAutoSelCond,
              O_OverTimeAutoSel => #AB_OverTimeAutoSel,
              O_HMISetCmd => #HMISetCmd,
              O_HMIResetCmd => #HMIResetCmd);
   END_IF;
END_REGION

REGION Network 6: **** 4.6 - Machine status - Indications **** Valve Animation for HMI
   // Valve Animation for HMI
